	100: (* Done *)
		bDone := (nErrorId = BACnet_ERR_NO_ERROR);
		(* release ADS buffer *)
		stBACnet_AdsBuffer.iLocked := 0;
		(* go idle *)
		_i := 0;

END_CASE

(* set error flag *)
bError 	:= nErrorId > BACnet_ERR_NO_ERROR;
bBusy 	:= _i > 0;
END_FUNCTION_BLOCK
ACTION _NextLogDatum:
_bNextDatum := (_pLrDatumList^.nEntrySize AND 16#80000000) = 16#80000000;
_cbTmpSize := 	(_F_BACnet_AlignedSize(_pLrDatumList^.nEntrySize) AND 16#7FFFFFFF)
			+	SIZEOF(_pLrDatumList^.nEntrySize)
			+	SIZEOF(_pLrDatumList^.reserved);
_pLrDatumList := _pLrDatumList + _cbTmpSize;
END_ACTION
ACTION _NextLogRecord:
_bNextRecord := ((_pLbRecordList^.nEntrySize AND 16#80000000) = 16#80000000);
_cbTmpSize := _F_BACnet_AlignedSize(_pLbRecordList^.nEntrySize AND 16#7FFFFFFF) + SIZEOF(_pLbRecordList^.nEntrySize) + SIZEOF(_pLbRecordList^.nSequence);
_pLbRecordList	:= _pLbRecordList + _cbTmpSize;
_cbTotalBuf := _cbTotalBuf + _cbTmpSize;
END_ACTION

(* POU FB_BACnet_ObjectNameProperty, ST *)
FUNCTION_BLOCK FB_BACnet_ObjectNameProperty
VAR_INPUT
	tObjectID			: T_BACnet_ObjectIdentifier := 16#FFFFFFFF;
	bAutoGet			: BOOL:=TRUE; (* TRUE = get data from property when ADS connection OR object ID changed *)
	bGet				: BOOL; (* FALSE --> TRUE = get data from property *)
END_VAR
VAR_IN_OUT
	stAdsConn			: ST_BACnet_AdsConnection;
END_VAR
VAR_OUTPUT
	bDone				: BOOL;
	bBusy				: BOOL;
	bError				: BOOL;
	nErrorId			: UINT;
	sText				: T_MaxString; (* Object name *)
END_VAR
VAR
	_fbReadProp		: FB_BACnet_ReadProp;
	_i				: INT;
	_rtrigGetSet	: R_TRIG;
	_nAdsReloadOld	: USINT;
	_tObjectIDOld	: T_BACnet_ObjectIdentifier := 16#FFFFFFFF;
	_StringExtDecode: FB_BACnet_StringExtDecode;
END_VAR
(* ADS read *)
_fbReadProp(
	BACnetDevicePort	:= stAdsConn.nAmsPort,
	bExecute			:= ,
	sNetId				:= stAdsConn.sAmsNetId,
	ObjectType			:= F_BACnet_GetObjType(tObjectID),
	PropertyID			:= BACnetPropertyIdentifier_ObjectName,
	DataType			:= BACnetDataType_CharacterStringExt,
	ObjectInstance		:= F_BACnet_GetObjInstance(tObjectID),
	ptrValue			:= ADR(sText),
	nLenValue			:= SIZEOF(sText)-1,
	bDone				=> ,
	bBusy				=> ,
	bError				=> ,
	nErrID				=> ,
	nProcessedLen		=> );

(* trigger start event *)
_rtrigGetSet(CLK:= bGet, Q=> );

(* state machine *)
CASE _i OF

	0: (* Idle *)
		IF		(		(		_rtrigGetSet.Q
							OR	(_nAdsReloadOld <> stAdsConn.nReload)
							OR	(_tObjectIDOld <> tObjectID)
						)
					AND	bAutoGet
				)
			OR	_rtrigGetSet.Q
		THEN
			IF (NOT stAdsConn.bValid) THEN
				(* ADS connection not valid *)
				nErrorId := BACnet_ERR_INVALID_ADS_CONN;
			ELSE
				nErrorId := BACnet_ERR_NO_ERROR;
				_i := 1;
				sText := '';
				(* remind ADS reload counter and parameter *)
				_nAdsReloadOld := stAdsConn.nReload;
				_tObjectIDOld := tObjectID;
			END_IF
			(* reset done flag *)
			bDone := FALSE;
		END_IF
		IF (NOT bGet) AND (NOT bAutoGet) THEN
			nErrorId := BACnet_ERR_NO_ERROR;
			bDone := FALSE;
		END_IF

	(* READ *)
	1: (* read object property data over ADS *)
		IF _fbReadProp.bExecute THEN
			IF _fbReadProp.bError THEN
				_i := 100;
				nErrorId := BACnet_ERR_ADS_Read;
				_fbReadProp.bExecute := FALSE;
			ELSIF (NOT _fbReadProp.bBusy) THEN
				_fbReadProp.bExecute := FALSE;
				(* decode property data *)
				_StringExtDecode(
					pChrStringExt	:= ADR(sText),
					nSize			:= _fbReadProp.nProcessedLen,
					pOutString		:= ADR(sText),
					bValid			=> ,
					bOverflow		=> ,
					nLength			=> ,
					eSrcEncoding	=> );
				(* check overflow flag *)
				IF _StringExtDecode.bOverflow THEN
					nErrorId := BACnet_ERR_ADS_BufferSize;
				END_IF
				(* DONE *)
				_i := 100;
			END_IF
		ELSE
			_fbReadProp.bExecute := TRUE;
		END_IF

	100: (* Done *)
		bDone := (nErrorId = BACnet_ERR_NO_ERROR);
		_i := 0;

END_CASE

(* set error flag *)
bError 	:= nErrorId > BACnet_ERR_NO_ERROR;
bBusy 	:= _i > 0;
END_FUNCTION_BLOCK

(* POU FB_BACnet_Loop, ST *)
FUNCTION_BLOCK FB_BACnet_Loop
VAR_INPUT
	fAccLimit		: REAL := 0.0; (* Setpoint acceleration limit positive and negative [1/s] *)
END_VAR
VAR_IN_OUT
	Device			: FB_BACnet_Device;
END_VAR
VAR_OUTPUT
	bReady			: BOOL;
	fSetPoint		: REAL;
	fControlledValue: REAL;
	fPresentValue	: REAL;
	fPropBand		: REAL; (* controller output in range of -100...100% in relation to Min.-/Max.-output *)
	bOverridden		: BOOL;
	bOutOfService	: BOOL;
	bFault			: BOOL;
	bInAlarm		: BOOL;
	bOpenLoop		: BOOL;
	bCommFailure	: BOOL;
	bOtherFault		: BOOL;
	bError			: BOOL;
	nErrorId		: UINT;
END_VAR
VAR
	_ControlledVariableValue AT%I*: REAL;	(* ~(BACnet_ControlledVariableValue :		: )
												(BACnet_ObjectType				: LOOP	: )	*)
	_Setpoint AT%I*:REAL;					(* ~(BACnet_Setpoint				:		: )	*)
	_ProportionalConstant AT%I*:REAL;		(* ~(BACnet_ProportionalConstant	:		: )	*)
	_IntegralConstant AT%I*:REAL;			(* ~(BACnet_IntegralConstant	 	:		: )	*)
	_DerivativeConstant AT%I*:REAL;			(* ~(BACnet_DerivativeConstant	 	:		: )	*)
	_MaximumOutput AT%I*:REAL;				(* ~(BACnet_MaximumOutput			:		: )	*)
	_MinimumOutput AT%I*:REAL;				(* ~(BACnet_MinimumOutput			:		: )	*)
	_Bias AT%I*:REAL;						(* ~(BACnet_Bias					:		: )	*)
	_PresentValueI AT%I*: REAL; 			(* ~(BACnet_PresentValue 			: 		: )	*)
	_StatusFlags AT%I*: WORD; 				(* ~(BACnet_StatusFlags 			: 		: )	*)
	_Reliability AT%I*: E_BACNETRELIABILITY;(* ~(BACNET_RELIABILITY 			:		: )	*)
	_ControlAction AT%I*:E_BACNETACTION;	(* ~(BACNET_ACTION				 	:		: )	*)
	_PresentValueQ AT%Q*: REAL;				(* ~(BACnet_PresentValue	 		:		: )	*)
	_StatusFlagsBits : ST_BACnet_StatusFlags;

	_sysTime	: GETCPUCOUNTER;
	_Time		: T_LARGE_INTEGER;
	_TimeOld	: T_LARGE_INTEGER;
	_cycleTime	: REAL;
	_PidControl : FB_BACnet_PidControl;
	_fbAccLimit : FB_BACnet_AccLimit;

	_nUpdateCount : UDINT := 0;
END_VAR
(* update server device *)
IF (Device._nUpdateCount = _nUpdateCount) THEN
	Device();
END_IF
(* remind current number of update counter *)
_nUpdateCount := Device._nUpdateCount;

(* determine cycle time *)
_TimeOld := _Time;
_sysTime(cpuCntLoDW=> _Time.dwLowPart, cpuCntHiDW=> _Time.dwHighPart);
_cycleTime := _F_BACnet_SysTimeDiff(In1:=_Time, In2:=_TimeOld);

(* check BitString format of StatusFlags --> if StatusFlags are less than 4, object isn't linked correctly *)
IF (_StatusFlags < 4) THEN
	(* wrong mapping *)
	nErrorId := BACnet_ERR_WRONG_MAPPING;
	bReady := FALSE;

ELSIF Device.bOperational THEN
	(* ready state *)
	bReady := TRUE;
	nErrorId := BACnet_ERR_NO_ERROR;

	(* decode status flags *)
	_StatusFlagsBits := F_BACnet_StatusFlags(_StatusFlags);

	(* copy states to output *)
	bOverridden := _StatusFlagsBits.overridden;
	bOutOfService := _StatusFlagsBits.out_of_service;
	bFault := _StatusFlagsBits.fault;
	bInAlarm := _StatusFlagsBits.in_alarm;
	bOpenLoop := (_Reliability = BACnetReliability_open_loop);
	bCommFailure := (_Reliability = BACnetReliability_communication_failure);
	bOtherFault := (_Reliability = BACnetReliability_unreliable_other);

	(* check reliability *)
	IF _Reliability <> BACnetReliability_no_fault_detected THEN
		_PidControl.bReset			:= TRUE;

	(* is set out of service? *)
	ELSIF _StatusFlagsBits.out_of_service THEN
		_PidControl.bReset			:= TRUE;

	(* decide the control action (direct or reverse) *)
	ELSIF _ControlAction = BACnetAction_direct THEN
		_PidControl.bReset			:= FALSE;
		_PidControl.fPresentValue	:= _ControlledVariableValue;
		_PidControl.fSetpoint		:= _Setpoint;

	ELSIF _ControlAction = BACnetAction_reverse THEN
		_PidControl.bReset			:= FALSE;
		_PidControl.fPresentValue	:= _Setpoint;
		_PidControl.fSetpoint		:= _ControlledVariableValue;

	ELSE
		(* unknown action *)
		_PidControl.bReset			:= TRUE;
	END_IF

	(* call PID control function block *)
	_PidControl(
		fCtrlCycleTime	:= _cycleTime,
		fBias			:= _Bias,
		fKp				:= _ProportionalConstant,
		fKi				:= _IntegralConstant,
		fKd				:= _DerivativeConstant,
		fTp				:= -1.0,
		fMaxOutput		:= _MaximumOutput,
		fMinOutput		:= _MinimumOutput,
		nErrorStatus	=>
	);
	_fbAccLimit.X := _PidControl.fY;

	(* set other outputs *)
	fSetPoint := _Setpoint;
	fPresentValue := _PresentValueI;
	fControlledValue := _ControlledVariableValue;
ELSE
	(* server device not ready, reset local ready also *)
	bReady := FALSE;
	nErrorId := BACnet_ERR_OPERATIONAL;
END_IF

(* limit present value *)
_fbAccLimit(X:= , Amax:= fAccLimit, Tcycle:= _cycleTime, Y=> _PresentValueQ, A=> );

(* calculate proportional band *)
IF (_MaximumOutput > 0.0) AND (_MinimumOutput >= 0.0) THEN
	fPropBand := ((_PresentValueQ - _MinimumOutput) / (_MaximumOutput - _MinimumOutput)) * 100.0;
ELSIF (_MaximumOutput <= 0.0) AND (_MinimumOutput < 0.0) THEN
	fPropBand := ((_PresentValueQ - _MaximumOutput) / (_MaximumOutput - _MinimumOutput)) * 100.0;
ELSIF (_PresentValueQ > 0.0) AND (_MaximumOutput > 0.0) THEN
	fPropBand := (_PresentValueQ / _MaximumOutput) * 100.0;
ELSIF (_PresentValueQ < 0.0) AND (_MinimumOutput < 0.0) THEN
	fPropBand := (_PresentValueQ / _MinimumOutput) * -100.0;
ELSE
	fPropBand := 0.0;
END_IF

(* set error flag *)
bError := (nErrorId <> BACnet_ERR_NO_ERROR);
END_FUNCTION_BLOCK

(* POU FB_BACnet_PidControl, ST *)
FUNCTION_BLOCK FB_BACnet_PidControl
VAR_INPUT
	(* controller input  *)
	fSetpoint				: REAL;	(* setpoint value *)
	fPresentValue			: REAL;	(* actual value *)
	(* reset flag *)
	bReset					: BOOL;
	(* controller values *)
	fCtrlCycleTime			: REAL; (* controller cycle time in seconds [s] *)

	fBias					: REAL; (* bias also active when reset is set to 1 *)
	fKp						: REAL;	(* proportional gain Kp	(P) *)
	fKi						: REAL; (* integral gain Ki (I) *)
	fKd						: REAL;	(* derivative gain Kd (D) *)
	fTp						: REAL := -1.0;	(* damping time Tp (PT1) [s] (fTp < 0 --> Tp = Kd / 10) *)

	(* maximum ratings *)
	fMaxOutput				: REAL;
	fMinOutput				: REAL;
END_VAR
VAR_OUTPUT
	fY						: REAL; (* controller output command *)
	nErrorStatus			: UINT; (* controller error output (0: no error; >0:error) *)
END_VAR
VAR
	(* Internal Variable *)
	_fE		: REAL;
	_fEOld	: REAL;
	_fYp	: REAL;
	_fYi	: REAL;
	_fYd	: REAL;
	_fbYd	: FB_BACnet_PT1;
END_VAR
(* preset error number *)
nErrorStatus	:= BACnet_ERR_NO_ERROR;

(* check cycle time parameter: (CycleTime > 0) *)
IF (fCtrlCycleTime <= 0.0) THEN
	nErrorStatus := BACnet_ERR_INVALID_CYCLETIME;
	bReset := TRUE;
END_IF;

(* check controller parameters: (Kp, Ki, Kd >= 0) *)
IF ((fKp < 0.0) OR (fKi < 0.0) OR (fKd < 0.0)) THEN
	nErrorStatus := BACnet_ERR_INVALID_PARAMETER;
	bReset := TRUE;
END_IF;

(* controller reset *)
IF bReset THEN
	(* reset internal and external variables *)
	_fEOld	:= 0.0;
	fY		:= MAX(MIN(fBias, fMaxOutput), fMinOutput);
	_fYi	:= 0.0;
	_fbYd(X:= 0.0, T:= 0.0, Y=> );
	RETURN;
END_IF

(* 3. save old variable *)
_fEOld := _fE;

(* 4. set error/deviation input *)
_fE := fSetpoint - fPresentValue;

(* 5. YP-part *)
_fYp := fKp * _fE;

(* 6. YI-part *)
IF (fKi = 0.0) THEN
	_fYi	:= 0.0;
ELSE
	_fYi := _fYi + (fKi * fCtrlCycleTime * _fE);
END_IF
IF (_fYi > fMaxOutput) THEN
	(* limit wind up positive *)
	_fYi := fMaxOutput;
ELSIF (_fYi < fMinOutput) THEN
	(* limit wind up negative *)
	_fYi := fMinOutput;
END_IF

(* 7. YD-part *)
IF (fTp < 0.0) THEN
	fTp := fKd / 10.0;
END_IF
_fYd := fKd * (_fE - _fEOld) / fCtrlCycleTime;
_fbYd(X:= _fYd, T:= fTp, Tcycle:= fCtrlCycleTime, Y=> );

(* 8. Ysum = YP + YI + YD + Bias and output *)
fY := _fYp + _fYi + _fbYd.Y + fBias;
fY := MAX(MIN(fY, fMaxOutput), fMinOutput);
END_FUNCTION_BLOCK

(* POU FB_BACnet_Loop_DRV, ST *)
FUNCTION_BLOCK FB_BACnet_Loop_DRV
VAR_IN_OUT
	Device	: FB_BACnet_Device;
END_VAR
VAR_OUTPUT
	bReady				: BOOL;
	fSetPoint			: REAL;
	fControlledValue	: REAL;
	fPresentValue		: REAL;
	bOverridden			: BOOL;
	bOutOfService		: BOOL;
	bFault				: BOOL;
	bInAlarm			: BOOL;
	bError				: BOOL;
	nErrorId			: UINT;
END_VAR
VAR
	_ControlledVariableValue AT%I*: REAL;	(* ~(BACnet_ControlledVariableValue :		: )
												(BACnet_ObjectType				: LOOP	: )
												(BACnet_EnableInternalLoopCtrl	: TRUE	: NOLINK,ENABLE) *)
	_Setpoint AT%I*:REAL;					(* ~(BACnet_Setpoint				:		: )	*)
	_PresentValue AT%I*: REAL; 				(* ~(BACnet_PresentValue 			: 		: )	*)
	_ObjectId AT%I*: DWORD;					(* ~(BACnet_ObjectIdentifier		:		: LINK) *)
	_StatusFlags AT%I*: WORD; 				(* ~(BACnet_StatusFlags 			: 		: )	*)
	_StatusFlagsBits : ST_BACnet_StatusFlags;
	_nUpdateCount : UDINT := 0;
END_VAR
(* update server device *)
IF (Device._nUpdateCount = _nUpdateCount) THEN
	Device();
END_IF
(* remind current number of update counter *)
_nUpdateCount := Device._nUpdateCount;

(* check BitString format of StatusFlags --> if StatusFlags are less than 4, object isn't linked correctly *)
IF (_StatusFlags < 4) THEN
	(* wrong mapping *)
	nErrorId := BACnet_ERR_WRONG_MAPPING;
	bReady := FALSE;

ELSIF Device.bOperational THEN
	(* ready state *)
	bReady := TRUE;
	nErrorId := BACnet_ERR_NO_ERROR;

	(* decode status flags *)
	_StatusFlagsBits := F_BACnet_StatusFlags(_StatusFlags);

	(* copy states to output *)
	bOverridden := _StatusFlagsBits.overridden;
	bOutOfService := _StatusFlagsBits.out_of_service;
	bFault := _StatusFlagsBits.fault;
	bInAlarm := _StatusFlagsBits.in_alarm;

	(* set other outputs *)
	fSetPoint := _Setpoint;
	fPresentValue := _PresentValue;
	fControlledValue := _ControlledVariableValue;
ELSE
	(* server device not ready, reset local ready also *)
	bReady := FALSE;
	nErrorId := BACnet_ERR_OPERATIONAL;
END_IF
(* set error flag *)
bError := (nErrorId <> BACnet_ERR_NO_ERROR);
END_FUNCTION_BLOCK

(* POU FB_BACnet_Loop_DRV_EX, ST *)
FUNCTION_BLOCK FB_BACnet_Loop_DRV_EX
VAR_IN_OUT
	Device	: FB_BACnet_Device;
END_VAR
VAR_OUTPUT
	bReady				: BOOL;
	fSetPoint			: REAL;
	fControlledValue	: REAL;
	fPresentValue		: REAL;
	fPropBand			: REAL; (* controller output in range of -100...100% in relation to Min.-/Max.-output *)
	bOverridden			: BOOL;
	bOutOfService		: BOOL;
	bFault				: BOOL;
	bInAlarm			: BOOL;
	bOpenLoop			: BOOL;
	bCommFailure		: BOOL;
	bOtherFault			: BOOL;
	eEventState			: E_BACNETEVENTSTATE;
	bAckedTrans_ToOffNormal : BOOL;
	bAckedTrans_ToFault		: BOOL;
	bAckedTrans_ToNormal	: BOOL;
	tObjectID			: T_BACnet_ObjectIdentifier := 16#FFFFFFFF;
	bError				: BOOL;
	nErrorId			: UINT;
END_VAR
VAR
	_ControlledVariableValue AT%I*: REAL;	(* ~(BACnet_ControlledVariableValue :		: )
												(BACnet_ObjectType				: LOOP	: )
												(BACnet_EnableInternalLoopCtrl	: TRUE	: NOLINK,ENABLE) *)
	_Setpoint AT%I*:REAL;					(* ~(BACnet_Setpoint				:		: )	*)
	_MaximumOutput AT%I*:REAL;				(* ~(BACnet_MaximumOutput			:		: )	*)
	_MinimumOutput AT%I*:REAL;				(* ~(BACnet_MinimumOutput			:		: )	*)
	_PresentValue AT%I*: REAL; 				(* ~(BACnet_PresentValue 			: 		: )	*)
	_ObjectId AT%I*: DWORD;					(* ~(BACnet_ObjectIdentifier		:		: LINK) *)
	_StatusFlags AT%I*: WORD; 				(* ~(BACnet_StatusFlags 			: 		: )	*)
	_AckedTransitions AT%I*:WORD;			(* ~(BACnet_AckedTransitions		:		: ) *)
	_EventState AT%I*: WORD; 				(* ~(BACnet_EventState 				:		: )	*)
	_Reliability AT%I*: E_BACNETRELIABILITY;(* ~(BACNET_RELIABILITY 			:		: )	*)
	_StatusFlagsBits : ST_BACnet_StatusFlags;
	_AckedTransBits : ST_BACnet_EventTransitionBits;
	_nUpdateCount : UDINT := 0;
END_VAR
(* update server device *)
IF (Device._nUpdateCount = _nUpdateCount) THEN
	Device();
END_IF
(* remind current number of update counter *)
_nUpdateCount := Device._nUpdateCount;

(* check BitString format of StatusFlags --> if StatusFlags are less than 4, object isn't linked correctly *)
IF (F_BACnet_GetObjType(_ObjectId) <> BACnetObjectType_Loop) THEN
	(* wrong mapping / invalid object ID *)
	IF _ObjectId = 0 THEN
		nErrorId := BACnet_ERR_WRONG_MAPPING;
	ELSE
		nErrorId := BACnet_ERR_INVALID_OBJECTID;
	END_IF
	bReady := FALSE;
	tObjectID := 16#FFFFFFFF;

ELSIF (_StatusFlags < 4) OR _AckedTransitions < 5 THEN
	(* wrong mapping *)
	nErrorId := BACnet_ERR_WRONG_MAPPING;
	bReady := FALSE;

ELSIF Device.bOperational THEN
	(* ready state *)
	bReady := TRUE;
	nErrorId := BACnet_ERR_NO_ERROR;

	(* decode status flags *)
	_StatusFlagsBits := F_BACnet_StatusFlags(_StatusFlags);
	_AckedTransBits	:= F_BACnet_EventTransitionFlags(_AckedTransitions);

	(* copy states to output *)
	bOverridden := _StatusFlagsBits.overridden;
	bOutOfService := _StatusFlagsBits.out_of_service;
	bFault := _StatusFlagsBits.fault;
	bInAlarm := _StatusFlagsBits.in_alarm;
	bOpenLoop := (_Reliability = BACnetReliability_open_loop);
	bCommFailure := (_Reliability = BACnetReliability_communication_failure);
	bOtherFault := (_Reliability = BACnetReliability_unreliable_other);
	bAckedTrans_ToOffNormal := _AckedTransBits.to_offnormal;
	bAckedTrans_ToFault := _AckedTransBits.to_fault;
	bAckedTrans_ToNormal := _AckedTransBits.to_normal;
	tObjectID := _ObjectId;
	eEventState := _EventState;

	(* calculate proportional band *)
	IF (_MaximumOutput > 0.0) AND (_MinimumOutput >= 0.0) THEN
		fPropBand := ((_PresentValue - _MinimumOutput) / (_MaximumOutput - _MinimumOutput)) * 100.0;
	ELSIF (_MaximumOutput <= 0.0) AND (_MinimumOutput < 0.0) THEN
		fPropBand := ((_PresentValue - _MaximumOutput) / (_MaximumOutput - _MinimumOutput)) * 100.0;
	ELSIF (_PresentValue > 0.0) AND (_MaximumOutput > 0.0) THEN
		fPropBand := (_PresentValue / _MaximumOutput) * 100.0;
	ELSIF (_PresentValue < 0.0) AND (_MinimumOutput < 0.0) THEN
		fPropBand := (_PresentValue / _MinimumOutput) * -100.0;
	ELSE
		fPropBand := 0.0;
	END_IF

	(* set other outputs *)
	fSetPoint := _Setpoint;
	fPresentValue := _PresentValue;
	fControlledValue := _ControlledVariableValue;
ELSE
	(* server device not ready, reset local ready also *)
	bReady := FALSE;
	nErrorId := BACnet_ERR_OPERATIONAL;
END_IF
(* set error flag *)
bError := (nErrorId <> BACnet_ERR_NO_ERROR);
END_FUNCTION_BLOCK

(* POU FB_BACnet_Loop_EX, ST *)
FUNCTION_BLOCK FB_BACnet_Loop_EX
VAR_INPUT
	bAutoTuning			: BOOL; (* Start autotuning of PID controller *)
	tTuningTimeout		: TIME := T#15m; (* Maximum runtime of tuning procedure [ms] *)
	eTuningMode			: E_BACNETPIDTUNINGMODE := BACnetPIDTuningMode_PI; (* optimize default PI controller *)
	fAccLimit			: REAL := 0.0; (* Setpoint acceleration limit positive and negative [1/s] *)
END_VAR
VAR_IN_OUT
	Device				: FB_BACnet_Device;
END_VAR
VAR_OUTPUT
	bReady				: BOOL;
	bTuningActive		: BOOL;
	bTuningWaitPV		: BOOL;
	bTuningWaitCV		: BOOL;
	bTuningDone			: BOOL;
	bTuningAborted		: BOOL;
	fSetPoint			: REAL;
	fControlledValue	: REAL;
	fPresentValue		: REAL;
	fPropBand			: REAL; (* controller output in range of -100...100% in relation to Min.-/Max.-output *)
	bOverridden			: BOOL;
	bOutOfService		: BOOL;
	bFault				: BOOL;
	bInAlarm			: BOOL;
	bOpenLoop			: BOOL;
	bCommFailure		: BOOL;
	bOtherFault			: BOOL;
	eEventState			: E_BACNETEVENTSTATE;
	bAckedTrans_ToOffNormal : BOOL;
	bAckedTrans_ToFault		: BOOL;
	bAckedTrans_ToNormal	: BOOL;
	tObjectID			: T_BACnet_ObjectIdentifier := 16#FFFFFFFF;
	bError				: BOOL;
	nErrorId			: UINT;
END_VAR
VAR
	_ControlledVariableValue AT%I*: REAL;	(* ~(BACnet_ControlledVariableValue :		: )
												(BACnet_ObjectType				: LOOP	: )	*)
	_Setpoint AT%I*:REAL;					(* ~(BACnet_Setpoint				:		: )	*)
	_ProportionalConstant AT%I*:REAL;		(* ~(BACnet_ProportionalConstant	:		: )	*)
	_IntegralConstant AT%I*:REAL;			(* ~(BACnet_IntegralConstant	 	:		: )	*)
	_DerivativeConstant AT%I*:REAL;			(* ~(BACnet_DerivativeConstant	 	:		: )	*)
	_MaximumOutput AT%I*:REAL;				(* ~(BACnet_MaximumOutput			:		: )	*)
	_MinimumOutput AT%I*:REAL;				(* ~(BACnet_MinimumOutput			:		: )	*)
	_Bias AT%I*:REAL;						(* ~(BACnet_Bias					:		: )	*)
	_PresentValueI AT%I*: REAL; 			(* ~(BACnet_PresentValue 			: 		: )	*)
	_Deadband AT%I*: REAL; 					(* ~(BACnet_Deadband	 			: 		: )	*)
	_ObjectId AT%I*: DWORD;					(* ~(BACnet_ObjectIdentifier		:		: LINK) *)
	_StatusFlags AT%I*: WORD; 				(* ~(BACnet_StatusFlags 			: 		: )	*)
	_AckedTransitions AT%I*:WORD;			(* ~(BACnet_AckedTransitions		:		: ) *)
	_EventState AT%I*: WORD; 				(* ~(BACnet_EventState 				:		: )	*)
	_Reliability AT%I*: E_BACNETRELIABILITY;(* ~(BACNET_RELIABILITY 			:		: )	*)
	_ControlAction AT%I*:E_BACNETACTION;	(* ~(BACNET_ACTION				 	:		: )	*)
	_PresentValueQ AT%Q*: REAL;				(* ~(BACnet_PresentValue	 		:		: )	*)
	_AckedTransBits : ST_BACnet_EventTransitionBits;
	_StatusFlagsBits : ST_BACnet_StatusFlags;

	_sysTime	: GETCPUCOUNTER;
	_Time		: T_LARGE_INTEGER;
	_TimeOld	: T_LARGE_INTEGER;
	_cycleTime	: REAL;
	_PidControl : FB_BACnet_PidControl;
	_AutoTuning : _FB_BACnet_PidTune;
	_iTuning	: INT;
	_WriteProp	: FB_BACnet_WriteProp;
	_fbAccLimit : FB_BACnet_AccLimit;
	_nUpdateCount : UDINT := 0;
END_VAR
(* update server device *)
IF (Device._nUpdateCount = _nUpdateCount) THEN
	Device();
END_IF
(* remind current number of update counter *)
_nUpdateCount := Device._nUpdateCount;

(* determine cycle time *)
_TimeOld := _Time;
_sysTime(cpuCntLoDW=> _Time.dwLowPart, cpuCntHiDW=> _Time.dwHighPart);
_cycleTime := _F_BACnet_SysTimeDiff(In1:=_Time, In2:=_TimeOld);

(* check BitString format of StatusFlags --> if StatusFlags are less than 4, object isn't linked correctly *)
IF (F_BACnet_GetObjType(_ObjectId) <> BACnetObjectType_Loop) THEN
	(* wrong mapping / invalid object ID *)
	IF _ObjectId = 0 THEN
		nErrorId := BACnet_ERR_WRONG_MAPPING;
	ELSE
		nErrorId := BACnet_ERR_INVALID_OBJECTID;
	END_IF
	bReady := FALSE;
	tObjectID := 16#FFFFFFFF;

ELSIF (_StatusFlags < 4) OR _AckedTransitions < 5 THEN
	(* wrong mapping *)
	nErrorId := BACnet_ERR_WRONG_MAPPING;
	bReady := FALSE;

ELSIF Device.bOperational THEN
	(* ready state *)
	bReady := TRUE;
	nErrorId := BACnet_ERR_NO_ERROR;

	(* decode status flags *)
	_StatusFlagsBits := F_BACnet_StatusFlags(_StatusFlags);
	_AckedTransBits	:= F_BACnet_EventTransitionFlags(_AckedTransitions);

	(* copy states to output *)
	bOverridden := _StatusFlagsBits.overridden;
	bOutOfService := _StatusFlagsBits.out_of_service;
	bFault := _StatusFlagsBits.fault;
	bInAlarm := _StatusFlagsBits.in_alarm;
	bOpenLoop := (_Reliability = BACnetReliability_open_loop);
	bCommFailure := (_Reliability = BACnetReliability_communication_failure);
	bOtherFault := (_Reliability = BACnetReliability_unreliable_other);
	bAckedTrans_ToOffNormal := _AckedTransBits.to_offnormal;
	bAckedTrans_ToFault := _AckedTransBits.to_fault;
	bAckedTrans_ToNormal := _AckedTransBits.to_normal;
	tObjectID := _ObjectId;
	eEventState := _EventState;

	(* check if auto tuning is active *)
	IF bTuningActive THEN
		_PidControl.bReset			:= TRUE;

	(* check reliability *)
	ELSIF _Reliability <> BACnetReliability_no_fault_detected THEN
		_PidControl.bReset			:= TRUE;

	(* is set out of service? *)
	ELSIF _StatusFlagsBits.out_of_service THEN
		_PidControl.bReset			:= TRUE;

	(* decide the control action (direct or reverse) *)
	ELSIF _ControlAction = BACnetAction_direct THEN
		_PidControl.bReset			:= FALSE;
		_PidControl.fPresentValue	:= _ControlledVariableValue;
		_PidControl.fSetpoint		:= _Setpoint;

	ELSIF _ControlAction = BACnetAction_reverse THEN
		_PidControl.bReset			:= FALSE;
		_PidControl.fPresentValue	:= _Setpoint;
		_PidControl.fSetpoint		:= _ControlledVariableValue;

	ELSE
		(* unknown action *)
		_PidControl.bReset			:= TRUE;
	END_IF

	(* call PID control function block *)
	_PidControl(
		fCtrlCycleTime	:= _cycleTime,
		fBias			:= _Bias,
		fKp				:= _ProportionalConstant,
		fKi				:= _IntegralConstant,
		fKd				:= _DerivativeConstant,
		fTp				:= -1.0,
		fMaxOutput		:= _MaximumOutput,
		fMinOutput		:= _MinimumOutput,
		nErrorStatus	=>
	);
	IF (_iTuning < 10) THEN
		_fbAccLimit.X := _PidControl.fY;
	END_IF

	(* set other outputs *)
	fSetPoint := _Setpoint;
	fPresentValue := _PresentValueI;
	fControlledValue := _ControlledVariableValue;
ELSE
	(* server device not ready, reset local ready also *)
	bReady := FALSE;
	nErrorId := BACnet_ERR_OPERATIONAL;
END_IF

(* write controller settings *)
_WriteProp.BACnetDevicePort:= Device.stAdsConn.nAmsPort;
_WriteProp.sNetId		:= Device.stAdsConn.sAmsNetId;
_WriteProp.ObjectType	:= BACnetObjectType_Loop;
_WriteProp.ObjectInstance:= F_BACnet_GetObjInstance(_ObjectId);

(* Autotuning function *)
CASE _iTuning OF
	0: (* Idle *)
		IF		bReady						(* object ready *)
			AND	(NOT _PidControl.bReset)	(* PID controller ready *)
			AND (tTuningTimeout > t#0ms)	(* timeout valid *)
			AND bAutoTuning					(* start flag *)
		THEN
			_iTuning := 5;
		END_IF
		_AutoTuning.bStart := FALSE;

	5:
		(* present_value low *)
		IF (_PresentValueI <= ((_MaximumOutput + _MinimumOutput) / 2.0) + _Bias) THEN
			_iTuning := 10;
		ELSIF (NOT bAutoTuning) THEN
			_iTuning := 0;
		END_IF

	10: (* setup *)
		_AutoTuning.fSetY	:= _MaximumOutput;
		_AutoTuning.tTimeout:= tTuningTimeout;
		_AutoTuning.fMinY	:= _MinimumOutput;
		_AutoTuning.fMaxY	:= _MaximumOutput;
		_AutoTuning.fDeadband:= _Deadband;
		_AutoTuning.eMode	:= eTuningMode;
		_iTuning := 20;

	20: (* wait busy *)
		_AutoTuning.bStart := TRUE;
		IF _AutoTuning.bAborted THEN
			_iTuning := 200;
		ELSIF _AutoTuning.bBusy THEN
			_iTuning := 30;
		END_IF

	30: (* wait done *)
		IF _AutoTuning.bAborted THEN
			_iTuning := 200;
		ELSIF _AutoTuning.bDone THEN
			_iTuning := 40;
		END_IF

	40: (* write properties *)
		IF Device.stAdsConn.bValid THEN
			_iTuning := 41;
			_WriteProp(bExecute := FALSE);
		ELSE
			_iTuning := 200;
		END_IF

	41: (* write Kp *)
		_WriteProp.DataType	:= BACnetDataType_Real;
		_WriteProp.ptrValue	:= ADR(_AutoTuning.fPID_Kp);
		_WriteProp.nLenValue:= SIZEOF(_AutoTuning.fPID_Kp);
		_WriteProp(
			bExecute := TRUE,
			PropertyID := BACnetPropertyIdentifier_ProportionalConstant);
		IF (NOT _WriteProp.bBusy) THEN
			IF (_WriteProp.bError) THEN
				_iTuning := 200;
			ELSE
				_iTuning := 42;
			END_IF
			_WriteProp(bExecute := FALSE);
		END_IF

	42: (* write Ki *)
		_WriteProp.DataType	:= BACnetDataType_Real;
		_WriteProp.ptrValue	:= ADR(_AutoTuning.fPID_Ki);
		_WriteProp.nLenValue:= SIZEOF(_AutoTuning.fPID_Ki);
		_WriteProp(
			bExecute := TRUE,
			PropertyID := BACnetPropertyIdentifier_IntegralConstant);
		IF (NOT _WriteProp.bBusy) THEN
			IF (_WriteProp.bError) THEN
				_iTuning := 200;
			ELSE
				_iTuning := 43;
			END_IF
			_WriteProp(bExecute := FALSE);
		END_IF

	43: (* write Kd *)
		_WriteProp.DataType	:= BACnetDataType_Real;
		_WriteProp.ptrValue	:= ADR(_AutoTuning.fPID_Kd);
		_WriteProp.nLenValue:= SIZEOF(_AutoTuning.fPID_Kd);
		_WriteProp(
			bExecute := TRUE,
			PropertyID := BACnetPropertyIdentifier_DerivativeConstant);
		IF (NOT _WriteProp.bBusy) THEN
			IF (_WriteProp.bError) THEN
				_iTuning := 200;
			ELSE
				_iTuning := 44;
			END_IF
			_WriteProp(bExecute := FALSE);
		END_IF

	44: (* write Action *)
		_WriteProp.DataType	:= BACnetDataType_Enumerated;
		_WriteProp.ptrValue	:= ADR(_AutoTuning.eAction);
		_WriteProp.nLenValue:= SIZEOF(_AutoTuning.eAction);
		_WriteProp(
			bExecute := TRUE,
			PropertyID := BACnetPropertyIdentifier_Action);
		IF (NOT _WriteProp.bBusy) THEN
			IF (_WriteProp.bError) THEN
				_iTuning := 200;
			ELSE
				_iTuning := 100;
			END_IF
			_WriteProp(bExecute := FALSE);
		END_IF


	100: (* done *)
		IF NOT bAutoTuning THEN
			_iTuning := 0;
		END_IF

	200: (* aborted *)
		IF NOT bAutoTuning THEN
			_iTuning := 0;
		END_IF

END_CASE

(* call auto tuning function block *)
_AutoTuning(
	bStart	:= ,
	bStop	:=	_StatusFlagsBits.out_of_service
			OR	(_Reliability <> BACnetReliability_no_fault_detected),
	fSetY	:= ,
	fDeadband	:= ,
	fX		:= _ControlledVariableValue,
	tTimeout:= ,
	fMinY	:= ,
	fMaxY	:= ,
	fCycleTime := _cycleTime,
	fY		:= _fbAccLimit.X,
	fPID_Kp	=> ,
	fPID_Ki	=> ,
	fPID_Kd	=> ,
	eAction => ,
	bSetY	=> ,
	bWaitY	=> ,
	bWaitX	=> ,
	bReady	=> ,
	bBusy	=> ,
	bDone	=> ,
	bAborted=> bTuningAborted,
	bTimeout=> );

(* set auto tuning state *)
bTuningWaitPV	:= (_iTuning = 5);
bTuningWaitCV	:= (_iTuning > 5 AND _iTuning <= 30);
bTuningAborted	:= (_iTuning = 200);
bTuningActive	:= (_iTuning > 0) AND (NOT bTuningAborted);
bTuningDone		:= (_iTuning = 100);
(* set error info *)
IF (bTuningActive OR bTuningAborted) THEN
	IF (NOT Device.stAdsConn.bValid) THEN
		nErrorId	:= BACnet_ERR_INVALID_ADS_CONN;
	ELSIF _WriteProp.bError THEN
		nErrorId	:= BACnet_ERR_ADS_Write;
	END_IF
END_IF

(* limit present value *)
_fbAccLimit(
	X	:= ,
	Amax:= fAccLimit,
	Tcycle:= _cycleTime,
	Y	=> _PresentValueQ,
	A	=> );

(* calculate proportional band *)
IF (_MaximumOutput > 0.0) AND (_MinimumOutput >= 0.0) THEN
	fPropBand := ((_PresentValueQ - _MinimumOutput) / (_MaximumOutput - _MinimumOutput)) * 100.0;
ELSIF (_MaximumOutput <= 0.0) AND (_MinimumOutput < 0.0) THEN
	fPropBand := ((_PresentValueQ - _MaximumOutput) / (_MaximumOutput - _MinimumOutput)) * 100.0;
ELSIF (_PresentValueQ > 0.0) AND (_MaximumOutput > 0.0) THEN
	fPropBand := (_PresentValueQ / _MaximumOutput) * 100.0;
ELSIF (_PresentValueQ < 0.0) AND (_MinimumOutput < 0.0) THEN
	fPropBand := (_PresentValueQ / _MinimumOutput) * -100.0;
ELSE
	fPropBand := 0.0;
END_IF

(* set error flag *)
bError := (nErrorId <> BACnet_ERR_NO_ERROR);
END_FUNCTION_BLOCK

(* POU FB_BACnet_MultiStateInput, ST *)
FUNCTION_BLOCK FB_BACnet_MultiStateInput
VAR_IN_OUT
	Device	: FB_BACnet_Device;
END_VAR
VAR_OUTPUT
	bReady			: BOOL;
	nPresentValue	: UDINT;
	bOverridden		: BOOL;
	bOutOfService	: BOOL;
	bFault			: BOOL;
	bInAlarm		: BOOL;
	bError			: BOOL;
	nErrorId		: UINT;
END_VAR
VAR
	_PresentValue AT%I*: UDINT; 	(* ~(BACnet_PresentValue 	:		: )
								   		(BACnet_ObjectType 		: MI	: )	*)
	_StatusFlags AT%I*: WORD; 		(* ~(BACnet_StatusFlags 	:		: )	*)
	_StatusFlagsBits : ST_BACnet_StatusFlags;

	_nUpdateCount : UDINT := 0;
END_VAR
(* update server device *)
IF (Device._nUpdateCount = _nUpdateCount) THEN
	Device();
END_IF
(* remind current number of update counter *)
_nUpdateCount := Device._nUpdateCount;

(* check BitString format of StatusFlags --> if StatusFlags are less than 4, object isn't linked correctly *)
IF (_StatusFlags < 4) THEN
	(* wrong mapping *)
	nErrorId := BACnet_ERR_WRONG_MAPPING;
	bReady := FALSE;

ELSIF Device.bOperational THEN
	(* ready state *)
	bReady := TRUE;
	nErrorId := BACnet_ERR_NO_ERROR;

	(* present value *)
	nPresentValue := _PresentValue;

	(* build bit states *)
	_StatusFlagsBits := F_BACnet_StatusFlags(_StatusFlags);

	(* copy states to output *)
	bOverridden := _StatusFlagsBits.overridden;
	bOutOfService := _StatusFlagsBits.out_of_service;
	bFault := _StatusFlagsBits.fault;
	bInAlarm := _StatusFlagsBits.in_alarm;

ELSE
	(* server device not ready, reset local ready also *)
	bReady := FALSE;
	nErrorId := BACnet_ERR_OPERATIONAL;
END_IF
(* set error flag *)
bError := (nErrorId <> BACnet_ERR_NO_ERROR);
END_FUNCTION_BLOCK

(* POU FB_BACnet_MultiStateInput_EX, ST *)
FUNCTION_BLOCK FB_BACnet_MultiStateInput_EX
VAR_IN_OUT
	Device				: FB_BACnet_Device;
END_VAR
VAR_OUTPUT
	bReady				: BOOL;
	nPresentValue		: UDINT;
	bOverridden			: BOOL;
	bOutOfService		: BOOL;
	bFault				: BOOL;
	bInAlarm			: BOOL;
	bOverRange			: BOOL;
	bUnderRange			: BOOL;
	bNoSensor			: BOOL;
	bOpenLoop			: BOOL;
	bShortedLoop		: BOOL;
	bMultiStateFault	: BOOL;
	bOtherFault			: BOOL;
	eEventState			: E_BACNETEVENTSTATE;
	bAckedTrans_ToOffNormal : BOOL;
	bAckedTrans_ToFault		: BOOL;
	bAckedTrans_ToNormal	: BOOL;
	nNbrOfStates		: UDINT;
	tObjectID			: T_BACnet_ObjectIdentifier := 16#FFFFFFFF;
	bError				: BOOL;
	nErrorId			: UINT;
END_VAR
VAR
	_PresentValue AT%I*: UDINT; 		(* ~(BACnet_PresentValue 	:		: )
								   			(BACnet_ObjectType 		: MI	: )	*)
	_NumberOfStates AT%I*: UDINT;		(* ~(BACnet_NumberOfStates	:		: )	*)
	_ObjectId AT%I*: DWORD;				(* ~(BACnet_ObjectIdentifier:		: LINK) *)
	_StatusFlags AT%I*: WORD; 			(* ~(BACnet_StatusFlags 	:		: )	*)
	_EventState AT%I*: WORD; 			(* ~(BACnet_EventState 		:		: )	*)
	_Reliability AT%I*: WORD; 			(* ~(BACnet_Reliability 	:		: )	*)
	_AckedTransitions AT%I*:WORD;		(* ~(BACnet_AckedTransitions:		: ) *)
	_AckedTransBits : ST_BACnet_EventTransitionBits;
	_nUpdateCount : UDINT := 0;
	_StatusFlagsBits : ST_BACnet_StatusFlags;
END_VAR
(* update server device *)
IF (Device._nUpdateCount = _nUpdateCount) THEN
	Device();
END_IF
(* remind current number of update counter *)
_nUpdateCount := Device._nUpdateCount;

(* check object type *)
IF (F_BACnet_GetObjType(_ObjectId) <> BACnetObjectType_MultiStateInput) THEN
	(* wrong mapping / invalid object ID *)
	IF _ObjectId = 0 THEN
		nErrorId := BACnet_ERR_WRONG_MAPPING;
	ELSE
		nErrorId := BACnet_ERR_INVALID_OBJECTID;
	END_IF
	bReady := FALSE;

ELSIF (_StatusFlags < 4) OR _AckedTransitions < 5 THEN
	(* wrong mapping *)
	nErrorId := BACnet_ERR_WRONG_MAPPING;
	bReady := FALSE;

ELSIF Device.bOperational THEN
	(* ready state *)
	bReady := TRUE;
	nErrorId := BACnet_ERR_NO_ERROR;

	(* present value *)
	nPresentValue := _PresentValue;

	(* build bit states *)
	_StatusFlagsBits := F_BACnet_StatusFlags(_StatusFlags);
	_AckedTransBits		:= F_BACnet_EventTransitionFlags(_AckedTransitions);

	(* copy states to output *)
	bOverridden := _StatusFlagsBits.overridden;
	bOutOfService := _StatusFlagsBits.out_of_service;
	bFault := _StatusFlagsBits.fault;
	bInAlarm := _StatusFlagsBits.in_alarm;
	bOverRange := (_Reliability = BACnetReliability_over_range);
	bUnderRange := (_Reliability = BACnetReliability_under_range);
	bNoSensor := (_Reliability = BACnetReliability_no_sensor);
	bOpenLoop := (_Reliability = BACnetReliability_open_loop);
	bShortedLoop := (_Reliability = BACnetReliability_shorted_loop);
	bMultiStateFault := (_Reliability = BACnetReliability_multi_state_fault);
	bOtherFault := (_Reliability = BACnetReliability_unreliable_other);
	bAckedTrans_ToOffNormal := _AckedTransBits.to_offnormal;
	bAckedTrans_ToFault := _AckedTransBits.to_fault;
	bAckedTrans_ToNormal := _AckedTransBits.to_normal;
	tObjectID := _ObjectId;

	(* convert enumeration *)
	eEventState := _EventState;

	(* number of states *)
	nNbrOfStates := _NumberOfStates;

ELSE
	(* server device not ready, reset local ready also *)
	bReady := FALSE;
	nErrorId := BACnet_ERR_OPERATIONAL;
END_IF
(* set error flag *)
bError := (nErrorId <> BACnet_ERR_NO_ERROR);
END_FUNCTION_BLOCK

(* POU FB_BACnet_MultiStateInput_RAW, ST *)
FUNCTION_BLOCK FB_BACnet_MultiStateInput_RAW
VAR_INPUT
	nRawIn				AT%Q*: DWORD; (* ~(BACnet_PresentValue : : ) *)
	bNoSensor		: BOOL;
	bOverRange		: BOOL;
	bUnderRange		: BOOL;
	bOpenLoop		: BOOL;
	bShortedLoop	: BOOL;
	bCommFailure	: BOOL;
	bOtherFault		: BOOL;
END_VAR
VAR_IN_OUT
	Device				: FB_BACnet_Device;
END_VAR
VAR_OUTPUT
	bReady				: BOOL;
	nPresentValue		: UDINT;
	bOverridden			: BOOL;
	bOutOfService		: BOOL;
	bFault				: BOOL;
	bInAlarm			: BOOL;
	bAckedTrans_ToOffNormal : BOOL;
	bAckedTrans_ToFault		: BOOL;
	bAckedTrans_ToNormal	: BOOL;
	nNbrOfStates		: UDINT;
	bError				: BOOL;
	nErrorId			: UINT;
END_VAR
VAR
	_Reliability AT%Q*: WORD := BACnetReliability_no_fault_detected;(* ~(BACnet_Reliability 	:		: )	*)
	_PresentValue AT%I*: UDINT; 		(* ~(BACnet_PresentValue 	:		: )
								   			(BACnet_ObjectType 		: MI	: )	*)
	_NumberOfStates AT%I*: UDINT;		(* ~(BACnet_NumberOfStates	:		: )	*)
	_ObjectId AT%I*: DWORD;				(* ~(BACnet_ObjectIdentifier:		: LINK) *)
	_StatusFlags AT%I*: WORD; 			(* ~(BACnet_StatusFlags 	:		: )	*)
	_AckedTransitions AT%I*:WORD;		(* ~(BACnet_AckedTransitions:		: ) *)
	_AckedTransBits : ST_BACnet_EventTransitionBits;
	_nUpdateCount : UDINT := 0;
	_StatusFlagsBits : ST_BACnet_StatusFlags;
END_VAR
(* update server device *)
IF (Device._nUpdateCount = _nUpdateCount) THEN
	Device();
END_IF
(* remind current number of update counter *)
_nUpdateCount := Device._nUpdateCount;

(* handle raw error *)
IF bNoSensor THEN
	_Reliability := BACnetReliability_no_sensor;
ELSIF bOverRange THEN
	_Reliability := BACnetReliability_over_range;
ELSIF bUnderRange THEN
	_Reliability := BACnetReliability_under_range;
ELSIF bOpenLoop THEN
	_Reliability := BACnetReliability_open_loop;
ELSIF bShortedLoop THEN
	_Reliability := BACnetReliability_shorted_loop;
ELSIF bCommFailure THEN
	_Reliability := BACnetReliability_communication_failure;
ELSIF bOtherFault THEN
	_Reliability := BACnetReliability_unreliable_other;
ELSE
	_Reliability := BACnetReliability_no_fault_detected;
END_IF

(* check object type *)
IF (F_BACnet_GetObjType(_ObjectId) <> BACnetObjectType_MultiStateInput) THEN
	(* wrong mapping / invalid object ID *)
	IF _ObjectId = 0 THEN
		nErrorId := BACnet_ERR_WRONG_MAPPING;
	ELSE
		nErrorId := BACnet_ERR_INVALID_OBJECTID;
	END_IF
	bReady := FALSE;

ELSIF (_StatusFlags < 4) OR _AckedTransitions < 5 THEN
	(* wrong mapping *)
	nErrorId := BACnet_ERR_WRONG_MAPPING;
	bReady := FALSE;

ELSIF Device.bOperational THEN
	(* ready state *)
	bReady := TRUE;
	nErrorId := BACnet_ERR_NO_ERROR;

	(* present value *)
	nPresentValue := _PresentValue;

	(* build bit states *)
	_StatusFlagsBits := F_BACnet_StatusFlags(_StatusFlags);
	_AckedTransBits		:= F_BACnet_EventTransitionFlags(_AckedTransitions);

	(* copy states to output *)
	bOverridden := _StatusFlagsBits.overridden;
	bOutOfService := _StatusFlagsBits.out_of_service;
	bFault := _StatusFlagsBits.fault;
	bInAlarm := _StatusFlagsBits.in_alarm;
	bAckedTrans_ToOffNormal := _AckedTransBits.to_offnormal;
	bAckedTrans_ToFault := _AckedTransBits.to_fault;
	bAckedTrans_ToNormal := _AckedTransBits.to_normal;

	(* number of states *)
	nNbrOfStates := _NumberOfStates;

ELSE
	(* server device not ready, reset local ready also *)
	bReady := FALSE;
	nErrorId := BACnet_ERR_OPERATIONAL;
END_IF
(* set error flag *)
bError := (nErrorId <> BACnet_ERR_NO_ERROR);
END_FUNCTION_BLOCK

(* POU FB_BACnet_MultiStateOutput, ST *)
FUNCTION_BLOCK FB_BACnet_MultiStateOutput
VAR_INPUT
	bEnablePV	: BOOL; (* enable present value with priority x in priority array, FALSE = priority x disable *)
	nPV			: UDINT; (* number for priority x, when input bEnablePV is TRUE *)
END_VAR
VAR_IN_OUT
	Device	: FB_BACnet_Device;
END_VAR
VAR_OUTPUT
	bReady			: BOOL;
	nPresentValue	: UDINT;
	bOverridden		: BOOL;
	bOutOfService	: BOOL;
	bFault			: BOOL;
	bInAlarm		: BOOL;
	nNbrOfStates	: UDINT;
	bError			: BOOL;
	nErrorId		: UINT;
END_VAR
VAR
	_PresentValue AT%I*: UDINT; 			(* ~(BACnet_PresentValue 		:		: )
								   				(BACnet_ObjectType			: MO	: )	*)
	_NumberOfStates AT%I*: UDINT;			(* ~(BACnet_NumberOfStates		:		: )	*)
	_StatusFlags AT%I*: WORD; 				(* ~(BACnet_StatusFlags			:		: )	*)
    _PresentValue_Priority12 AT%Q*: UDINT;	(* ~(BACnet_PresentValue_Priority12:	: )	*)
	_StatusFlagsBits : ST_BACnet_StatusFlags;
	_nUpdateCount : UDINT := 0;
END_VAR
(* update server device *)
IF (Device._nUpdateCount = _nUpdateCount) THEN
	Device();
END_IF
(* remind current number of update counter *)
_nUpdateCount := Device._nUpdateCount;

IF Device.bFirstCycle THEN
	(* first call of the server device since reboot/reset *)
	bReady := FALSE;
	_PresentValue_Priority12 := 0;

ELSIF (_StatusFlags < 4) THEN
	(* wrong mapping *)
	nErrorId := BACnet_ERR_WRONG_MAPPING;
	bReady := FALSE;

ELSIF Device.bOperational THEN
	(* ready state *)
	bReady := TRUE;
	nErrorId := BACnet_ERR_NO_ERROR;

	(* write into priority array *)
	IF bEnablePV THEN
		_PresentValue_Priority12	:= nPV;
	ELSE
		_PresentValue_Priority12	:= 0;
	END_IF

	(* present value *)
	nPresentValue := _PresentValue;

	(* build bit states *)
	_StatusFlagsBits := F_BACnet_StatusFlags(_StatusFlags);

	(* copy states to output *)
	bOverridden := _StatusFlagsBits.overridden;
	bOutOfService := _StatusFlagsBits.out_of_service;
	bFault := _StatusFlagsBits.fault;
	bInAlarm := _StatusFlagsBits.in_alarm;

	(* number of states *)
	nNbrOfStates := _NumberOfStates;

ELSE
	(* server device not ready, reset local ready also *)
	bReady := FALSE;
	nErrorId := BACnet_ERR_OPERATIONAL;
END_IF
(* set error flag *)
bError := (nErrorId <> BACnet_ERR_NO_ERROR);
END_FUNCTION_BLOCK

(* POU FB_BACnet_MultiStateOutput_ADS, ST *)
FUNCTION_BLOCK FB_BACnet_MultiStateOutput_ADS
VAR_INPUT
	bEnablePV			: BOOL;
	nPV					: UDINT; (* number for priority x, when input bEnablePV is TRUE *)
	bManual				: BOOL; (* FALSE --> TRUE: write present_value immediately, FALSE: only write present_value on-change, TRUE: write present_value on-change and when device turns operational *)
	ePriority			: E_BACNETPRIORITY := BACNETPRIORITY_12;
END_VAR
VAR_IN_OUT
	Device				: FB_BACnet_Device;
END_VAR
VAR_OUTPUT
	bReady				: BOOL;
	bPvDone				: BOOL; (* present_value written over ADS *)
	nPresentValue		: UDINT;
	bOverridden			: BOOL;
	bOutOfService		: BOOL;
	bFault				: BOOL;
	bInAlarm			: BOOL;
	nNbrOfStates		: UDINT;
	tObjectID			: T_BACnet_ObjectIdentifier := 16#FFFFFFFF;
	bError				: BOOL;
	nErrorId			: UINT;
	nAdsErrorId			: UDINT;
END_VAR
VAR
	_StatusFlags AT%I*: WORD; 				(* ~(BACnet_StatusFlags			:		: )	*)
	_PresentValue AT%I*: UDINT; 			(* ~(BACnet_PresentValue 		:		: )
								   				(BACnet_ObjectType			: MO	: )	*)
	_NumberOfStates AT%I*: UDINT;			(* ~(BACnet_NumberOfStates		:		: )	*)
	_ObjectId AT%I*: DWORD;					(* ~(BACnet_ObjectIdentifier	:		: LINK) *)
	_StatusFlagsBits : ST_BACnet_StatusFlags;
    _PresentValue_Ads : UDINT;
	_nUpdateCount : UDINT := 0;
	_WriteProp : FB_BACnet_WriteProp;
	_rtrigManual : R_TRIG;
	_bEnPvOld : BOOL;
	_nObjType : E_BACNETOBJECTTYPE;
END_VAR
(* update server device *)
IF (Device._nUpdateCount = _nUpdateCount) THEN
	Device();
END_IF
(* remind current number of update counter *)
_nUpdateCount := Device._nUpdateCount;

(* trigger on manual flag *)
_rtrigManual(CLK:= bManual, Q=> );

(* decode object type *)
_nObjType := F_BACnet_GetObjType(_ObjectId);

IF Device.bFirstCycle THEN
	(* first call of the server device since reboot/reset *)
	bReady := FALSE;
	bPvDone := FALSE;

ELSIF _nObjType <> BACnetObjectType_MultiStateOutput THEN
	(* wrong mapped object type *)
	nErrorId := BACnet_ERR_INVALID_OBJECTTYPE;
	bReady := FALSE;
	bPvDone := FALSE;

ELSIF (_StatusFlags < 4) THEN
	(* wrong mapping *)
	nErrorId := BACnet_ERR_WRONG_MAPPING;
	bReady := FALSE;
	bPvDone := FALSE;

ELSIF Device.bOperational THEN

	IF Device.stAdsConn.bValid THEN
		(* write present_value on manual trigger, on-change and on operational recover *)
		IF		_rtrigManual.Q
			OR	((nPV <> _PresentValue_Ads) AND bEnablePV)
			OR	((NOT bReady) AND bManual)
			OR	(bEnablePV <> _bEnPvOld)
		THEN
			_WriteProp.bExecute := TRUE;
			bPvDone := FALSE;
			(* write depending on enable state *)
			IF bEnablePV THEN
				_PresentValue_Ads := nPV;
			ELSE
				_PresentValue_Ads := 0;
			END_IF
			_bEnPvOld := bEnablePV;
		END_IF

		(* ready state *)
		IF (nAdsErrorId = 0) THEN
			bReady := TRUE;
			nErrorId := BACnet_ERR_NO_ERROR;
		END_IF

	ELSE
		(* invalid ADS connection *)
		bReady := FALSE;
		nErrorId := BACnet_ERR_INVALID_ADS_CONN;
		bPvDone := FALSE;
	END_IF

	(* present value *)
	nPresentValue := _PresentValue;

	(* build bit states *)
	_StatusFlagsBits := F_BACnet_StatusFlags(_StatusFlags);

	(* copy states to output *)
	bOverridden := _StatusFlagsBits.overridden;
	bOutOfService := _StatusFlagsBits.out_of_service;
	bFault := _StatusFlagsBits.fault;
	bInAlarm := _StatusFlagsBits.in_alarm;
	tObjectID := _ObjectId;

	(* number of states *)
	nNbrOfStates := _NumberOfStates;

ELSE
	(* server device not ready, reset local ready also *)
	bReady := FALSE;
	nErrorId := BACnet_ERR_OPERATIONAL;
	bPvDone := FALSE;
END_IF

(* call write property command *)
_WriteProp(
	BACnetDevicePort	:= Device.stAdsConn.nAmsPort,
	bExecute			:= ,
	sNetId				:= Device.stAdsConn.sAmsNetId,
	ObjectType			:= _nObjType,
	PropertyID			:= BACnetPropertyIdentifier_PresentValue,
	Priority			:= ePriority,
	DataType			:= BACnetDataType_UnsignedInteger,
	ObjectInstance		:= F_BACnet_GetObjInstance(_ObjectId),
	ptrValue			:= ADR(_PresentValue_Ads),
	nLenValue			:= SIZEOF(_PresentValue_Ads),
	bDone				=> ,
	bBusy				=> ,
	bError				=> ,
	nErrID				=> );

(* set done flag *)
IF _WriteProp.bExecute AND (NOT _WriteProp.bBusy) THEN
	(* check if command was finished with error *)
	IF _WriteProp.bError THEN
		bPvDone		:= FALSE;
		bReady		:= FALSE;
		nErrorId	:= BACnet_ERR_ADS_Write;
	ELSE
		(* successful written *)
		bPvDone		:= TRUE;
	END_IF
	nAdsErrorId := _WriteProp.nErrID;
	(* reset execution bit *)
	_WriteProp(bExecute := FALSE);
END_IF

(* set error flag *)
bError := (nErrorId <> BACnet_ERR_NO_ERROR) OR (nAdsErrorId <> 0);
END_FUNCTION_BLOCK

(* POU FB_BACnet_MultiStateOutput_EX, ST *)
FUNCTION_BLOCK FB_BACnet_MultiStateOutput_EX
VAR_INPUT
	bEnablePV			: BOOL; (* enable present value with priority x in priority array, FALSE = priority x disable *)
	nPV					: UDINT; (* number for priority x, when input bEnablePV is TRUE *)
END_VAR
VAR_IN_OUT
	Device				: FB_BACnet_Device;
END_VAR
VAR_OUTPUT
	bReady				: BOOL;
	nPresentValue		: UDINT;
	bOverridden			: BOOL;
	bOutOfService		: BOOL;
	bFault				: BOOL;
	bInAlarm			: BOOL;
	bNoOutput			: BOOL;
	bOpenLoop			: BOOL;
	bShortedLoop		: BOOL;
	bOtherFault			: BOOL;
	eEventState			: E_BACNETEVENTSTATE;
	bAckedTrans_ToOffNormal : BOOL;
	bAckedTrans_ToFault		: BOOL;
	bAckedTrans_ToNormal	: BOOL;
	nActivePrio			: UINT;
	nNbrOfStates		: UDINT;
	tObjectID			: T_BACnet_ObjectIdentifier := 16#FFFFFFFF;
	bError				: BOOL;
	nErrorId			: UINT;
END_VAR
VAR
	_PresentValue AT%I*: UDINT; 			(* ~(BACnet_PresentValue 		:		: )
								   				(BACnet_ObjectType			: MO	: )	*)
    _PresentValue_Priority12 AT%Q*: UDINT;	(* ~(BACnet_PresentValue_Priority12		:		: )	*)
	_ActivePriority AT%I*: UDINT; 			(* ~(BACnet_ActivePriority 		:		: )	*)
	_NumberOfStates AT%I*: UDINT;			(* ~(BACnet_NumberOfStates		:		: )	*)
	_ObjectId AT%I*: DWORD;					(* ~(BACnet_ObjectIdentifier	:		: LINK) *)
	_StatusFlags AT%I*: WORD; 				(* ~(BACnet_StatusFlags			:		: )	*)
	_EventState AT%I*: WORD;				(* ~(BACnet_EventState			:		: )	*)
	_Reliability AT%I*: WORD; 				(* ~(BACnet_Reliability			:		: )	*)
	_AckedTransitions AT%I*:WORD;			(* ~(BACnet_AckedTransitions	:		: ) *)
	_AckedTransBits : ST_BACnet_EventTransitionBits;
	_nUpdateCount : UDINT := 0;
	_StatusFlagsBits : ST_BACnet_StatusFlags;
END_VAR
(* update server device *)
IF (Device._nUpdateCount = _nUpdateCount) THEN
	Device();
END_IF
(* remind current number of update counter *)
_nUpdateCount := Device._nUpdateCount;

IF Device.bFirstCycle THEN
	(* first call of the server device since reboot/reset *)
	bReady := FALSE;
	_PresentValue_Priority12 := 0;

ELSIF (F_BACnet_GetObjType(_ObjectId) <> BACnetObjectType_MultiStateOutput) THEN
	(* wrong mapping / invalid object ID *)
	IF _ObjectId = 0 THEN
		nErrorId := BACnet_ERR_WRONG_MAPPING;
	ELSE
		nErrorId := BACnet_ERR_INVALID_OBJECTID;
	END_IF
	bReady := FALSE;

ELSIF (_StatusFlags < 4) OR _AckedTransitions < 5 THEN
	(* wrong mapping *)
	nErrorId := BACnet_ERR_WRONG_MAPPING;
	bReady := FALSE;

ELSIF Device.bOperational THEN
	(* ready state *)
	bReady := TRUE;
	nErrorId := BACnet_ERR_NO_ERROR;

	(* write into priority array *)
	IF bEnablePV THEN
		_PresentValue_Priority12	:= nPV;
	ELSE
		_PresentValue_Priority12	:= 0;
	END_IF

	(* present value *)
	nPresentValue := _PresentValue;

	(* build bit states *)
	_StatusFlagsBits := F_BACnet_StatusFlags(_StatusFlags);
	_AckedTransBits		:= F_BACnet_EventTransitionFlags(_AckedTransitions);

	(* copy states to output *)
	bOverridden := _StatusFlagsBits.overridden;
	bOutOfService := _StatusFlagsBits.out_of_service;
	bFault := _StatusFlagsBits.fault;
	bInAlarm := _StatusFlagsBits.in_alarm;
	bNoOutput := (_Reliability = BACnetReliability_no_output);
	bOpenLoop := (_Reliability = BACnetReliability_open_loop);
	bShortedLoop := (_Reliability = BACnetReliability_shorted_loop);
	bOtherFault := (_Reliability = BACnetReliability_unreliable_other);
	bAckedTrans_ToOffNormal := _AckedTransBits.to_offnormal;
	bAckedTrans_ToFault := _AckedTransBits.to_fault;
	bAckedTrans_ToNormal := _AckedTransBits.to_normal;
	tObjectID := _ObjectId;

	(* convert enumeration *)
	eEventState := _EventState;

	(* copy active priority *)
	nActivePrio := UDINT_TO_UINT(_ActivePriority);

	(* number of states *)
	nNbrOfStates := _NumberOfStates;

ELSE
	(* server device not ready, reset local ready also *)
	bReady := FALSE;
	nErrorId := BACnet_ERR_OPERATIONAL;
END_IF
(* set error flag *)
bError := (nErrorId <> BACnet_ERR_NO_ERROR);
END_FUNCTION_BLOCK

(* POU FB_BACnet_MultiStateOutput_RAW, ST *)
FUNCTION_BLOCK FB_BACnet_MultiStateOutput_RAW
VAR_INPUT
	bEnablePV			: BOOL; (* enable present value with priority x in priority array, FALSE = priority x disable *)
	nPV					: UDINT; (* number for priority x, when input bEnablePV is TRUE *)
	nFeedback			AT%Q*: DWORD; (* ~(BACnet_FeedbackValue : : ) *)
	bNoOutput			: BOOL;
	bOpenLoop			: BOOL;
	bShortedLoop		: BOOL;
	bCommFailure		: BOOL;
	bOtherFault			: BOOL;
END_VAR
VAR_IN_OUT
	Device				: FB_BACnet_Device;
END_VAR
VAR_OUTPUT
	bReady				: BOOL;
	nPresentValue		: UDINT;
	bOverridden			: BOOL;
	bOutOfService		: BOOL;
	bFault				: BOOL;
	bInAlarm			: BOOL;
	bAckedTrans_ToOffNormal : BOOL;
	bAckedTrans_ToFault		: BOOL;
	bAckedTrans_ToNormal	: BOOL;
	nNbrOfStates		: UDINT;
	bError				: BOOL;
	nErrorId			: UINT;
	nRawOut				AT%I*: DWORD;		(* ~(BACnet_PresentValue		:		: ) *)
END_VAR
VAR
    _PresentValue_Priority12 AT%Q*: UDINT;	(* ~(BACnet_PresentValue_Priority12:	: )
								   				(BACnet_ObjectType			: MO	: )	*)
	_Reliability AT%Q*: WORD := BACnetReliability_no_fault_detected;(* ~(BACnet_Reliability 	:		: )	*)
	_NumberOfStates AT%I*: UDINT;			(* ~(BACnet_NumberOfStates		:		: )	*)
	_ObjectId AT%I*: DWORD;					(* ~(BACnet_ObjectIdentifier	:		: LINK) *)
	_StatusFlags AT%I*: WORD; 				(* ~(BACnet_StatusFlags			:		: )	*)
	_AckedTransitions AT%I*:WORD;			(* ~(BACnet_AckedTransitions	:		: ) *)
	_AckedTransBits : ST_BACnet_EventTransitionBits;
	_nUpdateCount : UDINT := 0;
	_StatusFlagsBits : ST_BACnet_StatusFlags;
END_VAR
(* update server device *)
IF (Device._nUpdateCount = _nUpdateCount) THEN
	Device();
END_IF
(* remind current number of update counter *)
_nUpdateCount := Device._nUpdateCount;

(* handle raw error *)
IF bNoOutput THEN
	_Reliability := BACnetReliability_no_output;
ELSIF bOpenLoop THEN
	_Reliability := BACnetReliability_open_loop;
ELSIF bShortedLoop THEN
	_Reliability := BACnetReliability_shorted_loop;
ELSIF bCommFailure THEN
	_Reliability := BACnetReliability_communication_failure;
ELSIF bOtherFault THEN
	_Reliability := BACnetReliability_unreliable_other;
ELSE
	_Reliability := BACnetReliability_no_fault_detected;
END_IF

(* check object type *)
IF Device.bFirstCycle THEN
	(* first call of the server device since reboot/reset *)
	bReady := FALSE;
	_PresentValue_Priority12 := 0;

ELSIF (F_BACnet_GetObjType(_ObjectId) <> BACnetObjectType_MultiStateOutput) THEN
	(* wrong mapping / invalid object ID *)
	IF _ObjectId = 0 THEN
		nErrorId := BACnet_ERR_WRONG_MAPPING;
	ELSE
		nErrorId := BACnet_ERR_INVALID_OBJECTID;
	END_IF
	bReady := FALSE;

ELSIF (_StatusFlags < 4) OR _AckedTransitions < 5 THEN
	(* wrong mapping *)
	nErrorId := BACnet_ERR_WRONG_MAPPING;
	bReady := FALSE;

ELSIF Device.bOperational THEN
	(* ready state *)
	bReady := TRUE;
	nErrorId := BACnet_ERR_NO_ERROR;

	(* write into priority array *)
	IF bEnablePV THEN
		_PresentValue_Priority12	:= nPV;
	ELSE
		_PresentValue_Priority12	:= 0;
	END_IF

	(* present value *)
	nPresentValue := nRawOut;

	(* build bit states *)
	_StatusFlagsBits := F_BACnet_StatusFlags(_StatusFlags);
	_AckedTransBits		:= F_BACnet_EventTransitionFlags(_AckedTransitions);

	(* copy states to output *)
	bOverridden := _StatusFlagsBits.overridden;
	bOutOfService := _StatusFlagsBits.out_of_service;
	bFault := _StatusFlagsBits.fault;
	bInAlarm := _StatusFlagsBits.in_alarm;
	bAckedTrans_ToOffNormal := _AckedTransBits.to_offnormal;
	bAckedTrans_ToFault := _AckedTransBits.to_fault;
	bAckedTrans_ToNormal := _AckedTransBits.to_normal;

	(* number of states *)
	nNbrOfStates := _NumberOfStates;

ELSE
	(* server device not ready, reset local ready also *)
	bReady := FALSE;
	nErrorId := BACnet_ERR_OPERATIONAL;
END_IF
(* set error flag *)
bError := (nErrorId <> BACnet_ERR_NO_ERROR);
END_FUNCTION_BLOCK

(* POU FB_BACnet_MultiStateValue, ST *)
FUNCTION_BLOCK FB_BACnet_MultiStateValue
VAR_INPUT
	bEnablePV	: BOOL; (* enable present value with priority x in priority array, FALSE = priority x disable *)
	nPV			: UDINT; (* number for priority x, when input bEnablePV is TRUE *)
END_VAR
VAR_IN_OUT
	Device	: FB_BACnet_Device;
END_VAR
VAR_OUTPUT
	bReady			: BOOL;
	nPresentValue	: UDINT;
	bOverridden		: BOOL;
	bOutOfService	: BOOL;
	bFault			: BOOL;
	bInAlarm		: BOOL;
	nNbrOfStates	: UDINT;
	bError			: BOOL;
	nErrorId		: UINT;
END_VAR
VAR
	_PresentValue AT%I*: UDINT; 			(* ~(BACnet_PresentValue 		:		: )
								   				(BACnet_ObjectType 			: MV	: )	*)
	_NumberOfStates AT%I*: UDINT;			(* ~(BACnet_NumberOfStates		:		: )	*)
	_StatusFlags AT%I*: WORD; 				(* ~(BACnet_StatusFlags 		:		: )	*)
    _PresentValue_Priority12 AT%Q*: UDINT;	(* ~(BACnet_PresentValue_Priority12:	: )	*)
	_nUpdateCount : UDINT := 0;
	_StatusFlagsBits : ST_BACnet_StatusFlags;
END_VAR
(* update server device *)
IF (Device._nUpdateCount = _nUpdateCount) THEN
	Device();
END_IF
(* remind current number of update counter *)
_nUpdateCount := Device._nUpdateCount;

IF Device.bFirstCycle THEN
	(* first call of the server device since reboot/reset *)
	bReady := FALSE;
	_PresentValue_Priority12 := 0;

ELSIF (_StatusFlags < 4) THEN
	(* wrong mapping *)
	nErrorId := BACnet_ERR_WRONG_MAPPING;
	bReady := FALSE;

ELSIF Device.bOperational THEN
	(* ready state *)
	bReady := TRUE;
	nErrorId := BACnet_ERR_NO_ERROR;

	(* write into priority array *)
	IF bEnablePV THEN
		_PresentValue_Priority12	:= nPV;
	ELSE
		_PresentValue_Priority12	:= 0;
	END_IF

	(* present value *)
	nPresentValue := _PresentValue;

	(* build bit states *)
	_StatusFlagsBits := F_BACnet_StatusFlags(_StatusFlags);

	(* copy states to output *)
	bOverridden := _StatusFlagsBits.overridden;
	bOutOfService := _StatusFlagsBits.out_of_service;
	bFault := _StatusFlagsBits.fault;
	bInAlarm := _StatusFlagsBits.in_alarm;

	(* number of states *)
	nNbrOfStates := _NumberOfStates;

ELSE
	(* server device not ready, reset local ready also *)
	bReady := FALSE;
	nErrorId := BACnet_ERR_OPERATIONAL;
END_IF
(* set error flag *)
bError := (nErrorId <> BACnet_ERR_NO_ERROR);
END_FUNCTION_BLOCK

(* POU FB_BACnet_MultiStateValue_ADS, ST *)
FUNCTION_BLOCK FB_BACnet_MultiStateValue_ADS
VAR_INPUT
	bEnablePV			: BOOL;
	nPV					: UDINT; (* number for priority x, when input bEnablePV is TRUE *)
	bManual				: BOOL; (* FALSE --> TRUE: write present_value immediately, FALSE: only write present_value on-change, TRUE: write present_value on-change and when device turns operational *)
	ePriority			: E_BACNETPRIORITY := BACNETPRIORITY_12;
END_VAR
VAR_IN_OUT
	Device				: FB_BACnet_Device;
END_VAR
VAR_OUTPUT
	bReady				: BOOL;
	bPvDone				: BOOL; (* present_value written over ADS *)
	nPresentValue		: UDINT;
	bOverridden			: BOOL;
	bOutOfService		: BOOL;
	bFault				: BOOL;
	bInAlarm			: BOOL;
	nNbrOfStates		: UDINT;
	tObjectID			: T_BACnet_ObjectIdentifier := 16#FFFFFFFF;
	bError				: BOOL;
	nErrorId			: UINT;
	nAdsErrorId			: UDINT;
END_VAR
VAR
	_StatusFlags AT%I*: WORD; 				(* ~(BACnet_StatusFlags 	:		: )	*)
	_PresentValue AT%I*: UDINT; 			(* ~(BACnet_PresentValue 	:		: )
								   				(BACnet_ObjectType 		: MV	: )	*)
	_NumberOfStates AT%I*: UDINT;			(* ~(BACnet_NumberOfStates	:		: )	*)
	_ObjectId AT%I*: DWORD;					(* ~(BACnet_ObjectIdentifier:		: LINK) *)
	_StatusFlagsBits : ST_BACnet_StatusFlags;
    _PresentValue_Ads : UDINT;
	_nUpdateCount : UDINT := 0;
	_WriteProp : FB_BACnet_WriteProp;
	_rtrigManual : R_TRIG;
	_bEnPvOld : BOOL;
	_nObjType : E_BACNETOBJECTTYPE;
END_VAR
(* update server device *)
IF (Device._nUpdateCount = _nUpdateCount) THEN
	Device();
END_IF
(* remind current number of update counter *)
_nUpdateCount := Device._nUpdateCount;

(* trigger on manual flag *)
_rtrigManual(CLK:= bManual, Q=> );

(* decode object type *)
_nObjType := F_BACnet_GetObjType(_ObjectId);

IF Device.bFirstCycle THEN
	(* first call of the server device since reboot/reset *)
	bReady := FALSE;
	bPvDone := FALSE;

ELSIF _nObjType <> BACnetObjectType_MultiStateValue THEN
	(* wrong mapped object type *)
	nErrorId := BACnet_ERR_INVALID_OBJECTTYPE;
	bReady := FALSE;
	bPvDone := FALSE;

ELSIF (_StatusFlags < 4) THEN
	(* wrong mapping *)
	nErrorId := BACnet_ERR_WRONG_MAPPING;
	bReady := FALSE;
	bPvDone := FALSE;

ELSIF Device.bOperational THEN

	IF Device.stAdsConn.bValid THEN
		(* write present_value on manual trigger, on-change and on operational recover *)
		IF		_rtrigManual.Q
			OR	((nPV <> _PresentValue_Ads) AND bEnablePV)
			OR	((NOT bReady) AND bManual)
			OR	(bEnablePV <> _bEnPvOld)
		THEN
			_WriteProp.bExecute := TRUE;
			bPvDone := FALSE;
			(* write depending on enable state *)
			IF bEnablePV THEN
				_PresentValue_Ads := nPV;
			ELSE
				_PresentValue_Ads := 0;
			END_IF
			_bEnPvOld := bEnablePV;
		END_IF

		(* ready state *)
		IF (nAdsErrorId = 0) THEN
			bReady := TRUE;
			nErrorId := BACnet_ERR_NO_ERROR;
		END_IF

	ELSE
		(* invalid ADS connection *)
		bReady := FALSE;
		nErrorId := BACnet_ERR_INVALID_ADS_CONN;
		bPvDone := FALSE;
	END_IF

	(* present value *)
	nPresentValue := _PresentValue;

	(* build bit states *)
	_StatusFlagsBits := F_BACnet_StatusFlags(_StatusFlags);

	(* copy states to output *)
	bOverridden := _StatusFlagsBits.overridden;
	bOutOfService := _StatusFlagsBits.out_of_service;
	bFault := _StatusFlagsBits.fault;
	bInAlarm := _StatusFlagsBits.in_alarm;
	tObjectID := _ObjectId;

	(* number of states *)
	nNbrOfStates := _NumberOfStates;

ELSE
	(* server device not ready, reset local ready also *)
	bReady := FALSE;
	nErrorId := BACnet_ERR_OPERATIONAL;
	bPvDone := FALSE;
END_IF

(* call write property command *)
_WriteProp(
	BACnetDevicePort	:= Device.stAdsConn.nAmsPort,
	bExecute			:= ,
	sNetId				:= Device.stAdsConn.sAmsNetId,
	ObjectType			:= _nObjType,
	PropertyID			:= BACnetPropertyIdentifier_PresentValue,
	Priority			:= ePriority,
	DataType			:= BACnetDataType_UnsignedInteger,
	ObjectInstance		:= F_BACnet_GetObjInstance(_ObjectId),
	ptrValue			:= ADR(_PresentValue_Ads),
	nLenValue			:= SIZEOF(_PresentValue_Ads),
	bDone				=> ,
	bBusy				=> ,
	bError				=> ,
	nErrID				=> );

(* set done flag *)
IF _WriteProp.bExecute AND (NOT _WriteProp.bBusy) THEN
	(* check if command was finished with error *)
	IF _WriteProp.bError THEN
		bPvDone		:= FALSE;
		bReady		:= FALSE;
		nErrorId	:= BACnet_ERR_ADS_Write;
	ELSE
		(* successful written *)
		bPvDone		:= TRUE;
	END_IF
	nAdsErrorId := _WriteProp.nErrID;
	(* reset execution bit *)
	_WriteProp(bExecute := FALSE);
END_IF

(* set error flag *)
bError := (nErrorId <> BACnet_ERR_NO_ERROR) OR (nAdsErrorId <> 0);
END_FUNCTION_BLOCK

(* POU FB_BACnet_MultiStateValue_EX, ST *)
FUNCTION_BLOCK FB_BACnet_MultiStateValue_EX
VAR_INPUT
	bEnablePV			: BOOL; (* enable present value with priority x in priority array, FALSE = priority x disable *)
	nPV					: UDINT; (* number for priority x, when input bEnablePV is TRUE *)
END_VAR
VAR_IN_OUT
	Device				: FB_BACnet_Device;
END_VAR
VAR_OUTPUT
	bReady				: BOOL;
	nPresentValue		: UDINT;
	bOverridden			: BOOL;
	bOutOfService		: BOOL;
	bFault				: BOOL;
	bInAlarm			: BOOL;
	bMultiStateFault	: BOOL;
	bOtherFault			: BOOL;
	eEventState			: E_BACNETEVENTSTATE;
	bAckedTrans_ToOffNormal : BOOL;
	bAckedTrans_ToFault		: BOOL;
	bAckedTrans_ToNormal	: BOOL;
	nActivePrio			: UINT;
	nNbrOfStates		: UDINT;
	tObjectID			: T_BACnet_ObjectIdentifier := 16#FFFFFFFF;
	bError				: BOOL;
	nErrorId			: UINT;
END_VAR
VAR
	_PresentValue AT%I*: UDINT; 			(* ~(BACnet_PresentValue 	:		: )
								   				(BACnet_ObjectType 		: MV	: )	*)
    _PresentValue_Priority12 AT%Q*: UDINT;	(* ~(BACnet_PresentValue_Priority12	:		: )	*)
	_ActivePriority AT%I*: UDINT; 			(* ~(BACnet_ActivePriority 	:		: )	*)
	_NumberOfStates AT%I*: UDINT;			(* ~(BACnet_NumberOfStates	:		: )	*)
	_ObjectId AT%I*: DWORD;					(* ~(BACnet_ObjectIdentifier:		: LINK) *)
	_StatusFlags AT%I*: WORD; 				(* ~(BACnet_StatusFlags 	:		: )	*)
	_EventState AT%I*: WORD;				(* ~(BACnet_EventState 		:		: )	*)
	_Reliability AT%I*: WORD;				(* ~(BACnet_Reliability 	:		: )	*)
	_AckedTransitions AT%I*:WORD;			(* ~(BACnet_AckedTransitions:		: ) *)
	_AckedTransBits : ST_BACnet_EventTransitionBits;
	_StatusFlagsBits : ST_BACnet_StatusFlags;
	_nUpdateCount : UDINT := 0;
END_VAR
(* update server device *)
IF (Device._nUpdateCount = _nUpdateCount) THEN
	Device();
END_IF
(* remind current number of update counter *)
_nUpdateCount := Device._nUpdateCount;

IF Device.bFirstCycle THEN
	(* first call of the server device since reboot/reset *)
	bReady := FALSE;
	_PresentValue_Priority12 := 0;

ELSIF (F_BACnet_GetObjType(_ObjectId) <> BACnetObjectType_MultiStateValue) THEN
	(* wrong mapping / invalid object ID *)
	IF _ObjectId = 0 THEN
		nErrorId := BACnet_ERR_WRONG_MAPPING;
	ELSE
		nErrorId := BACnet_ERR_INVALID_OBJECTID;
	END_IF
	bReady := FALSE;

ELSIF (_StatusFlags < 4) OR _AckedTransitions < 5 THEN
	(* wrong mapping *)
	nErrorId := BACnet_ERR_WRONG_MAPPING;
	bReady := FALSE;

ELSIF Device.bOperational THEN
	(* ready state *)
	bReady := TRUE;
	nErrorId := BACnet_ERR_NO_ERROR;

	(* write into priority array *)
	IF bEnablePV THEN
		_PresentValue_Priority12	:= nPV;
	ELSE
		_PresentValue_Priority12	:= 0;
	END_IF

	(* present value *)
	nPresentValue := _PresentValue;

	(* build bit states *)
	_StatusFlagsBits := F_BACnet_StatusFlags(_StatusFlags);
	_AckedTransBits		:= F_BACnet_EventTransitionFlags(_AckedTransitions);

	(* copy states to output *)
	bOverridden := _StatusFlagsBits.overridden;
	bOutOfService := _StatusFlagsBits.out_of_service;
	bFault := _StatusFlagsBits.fault;
	bInAlarm := _StatusFlagsBits.in_alarm;
	bMultiStateFault := (_Reliability = BACnetReliability_multi_state_fault);
	bOtherFault := (_Reliability = BACnetReliability_unreliable_other);
	bAckedTrans_ToOffNormal := _AckedTransBits.to_offnormal;
	bAckedTrans_ToFault := _AckedTransBits.to_fault;
	bAckedTrans_ToNormal := _AckedTransBits.to_normal;
	tObjectID := _ObjectId;

	(* convert enumeration *)
	eEventState := _EventState;

	(* copy active priority *)
	nActivePrio := UDINT_TO_UINT(_ActivePriority);

	(* number of states *)
	nNbrOfStates := _NumberOfStates;

ELSE
	(* server device not ready, reset local ready also *)
	bReady := FALSE;
	nErrorId := BACnet_ERR_OPERATIONAL;
END_IF
(* set error flag *)
bError := (nErrorId <> BACnet_ERR_NO_ERROR);
END_FUNCTION_BLOCK

(* POU FB_BACnet_NotificationClass, ST *)
FUNCTION_BLOCK FB_BACnet_NotificationClass
VAR_IN_OUT
	Device	: FB_BACnet_Device;
END_VAR
VAR_OUTPUT
	bReady			: BOOL;
	bError			: BOOL;
	nErrorId		: UINT;
END_VAR
VAR
	_ObjectId AT%I* : DWORD;					(* ~(BACnet_ObjectIdentifier:		: LINK)
													(BACnet_ObjectType		:	NC	: ) *)
	_nUpdateCount	: UDINT := 0;
END_VAR
(* update server device *)
IF (Device._nUpdateCount = _nUpdateCount) THEN
	Device();
END_IF
(* remind current number of update counter *)
_nUpdateCount := Device._nUpdateCount;

IF Device.bOperational THEN
	(* ready state *)
	bReady := TRUE;
	nErrorId := BACnet_ERR_NO_ERROR;
ELSE
	(* server device not ready, reset local ready also *)
	bReady := FALSE;
	nErrorId := BACnet_ERR_OPERATIONAL;
END_IF
(* set error flag *)
bError := (nErrorId <> BACnet_ERR_NO_ERROR);
END_FUNCTION_BLOCK

(* POU FB_BACnet_NotificationClass_EX, ST *)
FUNCTION_BLOCK FB_BACnet_NotificationClass_EX
VAR_IN_OUT
	Device				: FB_BACnet_Device;
END_VAR
VAR_OUTPUT
	bReady				: BOOL;
	tObjectID			: T_BACnet_ObjectIdentifier := 16#FFFFFFFF;
	bError				: BOOL;
	nErrorId			: UINT;
END_VAR
VAR
	_ObjectId AT%I* : DWORD;					(* ~(BACnet_ObjectIdentifier:		: LINK)
													(BACnet_ObjectType		:	NC	: ) *)
	_nUpdateCount	: UDINT := 0;
END_VAR
(* update server device *)
IF (Device._nUpdateCount = _nUpdateCount) THEN
	Device();
END_IF
(* remind current number of update counter *)
_nUpdateCount := Device._nUpdateCount;

IF (F_BACnet_GetObjType(_ObjectId) <> BACnetObjectType_NotificationClass) THEN
	(* wrong mapping / invalid object ID *)
	IF _ObjectId = 0 THEN
		nErrorId := BACnet_ERR_WRONG_MAPPING;
	ELSE
		nErrorId := BACnet_ERR_INVALID_OBJECTID;
	END_IF
	bReady := FALSE;
	tObjectID := 16#FFFFFFFF;

ELSIF Device.bOperational THEN
	(* ready state *)
	bReady := TRUE;
	nErrorId := BACnet_ERR_NO_ERROR;
	tObjectID := _ObjectId;

ELSE
	(* server device not ready, reset local ready also *)
	bReady := FALSE;
	nErrorId := BACnet_ERR_OPERATIONAL;
END_IF
(* set error flag *)
bError := (nErrorId <> BACnet_ERR_NO_ERROR);
END_FUNCTION_BLOCK

(* POU FB_BACnet_NotificationSinkDelEntry, ST *)
FUNCTION_BLOCK FB_BACnet_NotificationSinkDelEntry
VAR_INPUT
	bExecute	: BOOL;
	nIndex		: UDINT;
	sNetId		: T_AmsNetId;
	nPort		: T_AmsPort;
	tTimeout	: TIME := BACnet_ADSTimeOut;
END_VAR
VAR_OUTPUT
	bBusy		: BOOL;
	bEmpty		: BOOL;
	bError		: BOOL;
	nErrorId	: UDINT;
END_VAR
VAR
	_AdsReadClient	: ADSREAD;
END_VAR
	_AdsReadClient(
		NETID	:= sNetId,
		PORT	:= nPort,
		IDXGRP	:= 16#5,
		IDXOFFS	:= nIndex,
		LEN		:= 0,
		DESTADDR:= 0,
		READ	:= bExecute,
		TMOUT	:= tTimeout,
		BUSY	=> bBusy,
		ERR		=> bError,
		ERRID	=> nErrorId);

	bEmpty := ((UDINT_TO_DWORD(_AdsReadClient.ERRID) AND 16#FFF) = 16#703);
END_FUNCTION_BLOCK

(* POU FB_BACnet_ObjectListProperty, ST *)
FUNCTION_BLOCK FB_BACnet_ObjectListProperty
VAR_INPUT
	bAutoGet			: BOOL:=TRUE; (* TRUE = get data from property when ADS connection OR object ID changed *)
	bGet				: BOOL; (* FALSE --> TRUE = get data from property *)
	bTypeFilter			: BOOL; (* activate input "eObjectTypeFilter" *)
	eObjType			: E_BACnetObjectType; (* select the object type that is scanned *)
END_VAR
VAR_IN_OUT
	stAdsConn			: ST_BACnet_AdsConnection;
END_VAR
VAR_OUTPUT
	bDone				: BOOL;
	bBusy				: BOOL;
	bError				: BOOL;
	nErrorId			: UINT;
	stObjIDList			: ST_BACnet_ObjectIdentifierList;
END_VAR
VAR
	_fbReadProp			: FB_BACnet_ReadProp;
	_i					: INT;
	_cbPropSize			: UDINT;
	_cbMemCpy			: UDINT;
	_nEntryCount		: UDINT;
	_iScan				: UDINT;
	_pEntry				: POINTER TO T_BACnet_ObjectIdentifier := 16#FFFFFFFF;
	_cbAdsBuf			: UDINT;
	_rtrigGetSet		: R_TRIG;
	_nAdsReloadOld		: USINT;
	_bUseObjTypeFilterOld: BOOL;
	_eObjTypeFilterOld	: E_BACnetObjectType;
	_nDeviceIdOld		: DWORD := 16#FFFFFFFF;
END_VAR
(* ADS read *);
_fbReadProp(
	BACnetDevicePort	:= stAdsConn.nAmsPort,
	bExecute			:= ,
	ObjectInstance		:= F_BACnet_GetObjInstance(stAdsConn.nDeviceId),
	ObjectType			:= BACnetObjectType_Device,
	sNetId				:= stAdsConn.sAmsNetId,
	PropertyID			:= BACnetPropertyIdentifier_ObjectList,
	DataType			:= BACnetDataType_ObjectIdentifierArr,
	ptrValue			:= ADR(stBACnet_AdsBuffer.arrData),
	nLenValue			:= SIZEOF(stBACnet_AdsBuffer.arrData),
	bDone				=> ,
	bBusy				=> ,
	bError				=> ,
	nErrID				=> ,
	nProcessedLen		=> );

(* trigger start event *)
_rtrigGetSet(CLK:= bGet, Q=> );

(* state machine *)
CASE _i OF

	0: (* Idle *)
		IF		(		(
								(_nAdsReloadOld <> stAdsConn.nReload)
							OR	(_bUseObjTypeFilterOld <> bTypeFilter)
							OR	((_eObjTypeFilterOld <> eObjType) AND bTypeFilter)
							OR	(_nDeviceIdOld <> stAdsConn.nDeviceId)
						)
					AND	bAutoGet
				)
			OR	_rtrigGetSet.Q
		THEN
			IF (NOT stAdsConn.bValid) THEN
				(* ADS connection not valid *)
				nErrorId := BACnet_ERR_INVALID_ADS_CONN;
			ELSE
				nErrorId := BACnet_ERR_NO_ERROR;
				_i := 1;
				(* remind ADS reload counter and parameter *)
				_nAdsReloadOld := stAdsConn.nReload;
				_bUseObjTypeFilterOld := bTypeFilter;
				_eObjTypeFilterOld := eObjType;
				_nDeviceIdOld := stAdsConn.nDeviceId;
			END_IF
			(* reset done flag *)
			bDone := FALSE;
		END_IF
		IF (NOT bGet) AND (NOT bAutoGet) THEN
			nErrorId := BACnet_ERR_NO_ERROR;
			bDone := FALSE;
		END_IF

	(* READ *)
	1: (* read object property data via ADS *)
		IF TestAndSet(stBACnet_AdsBuffer.bTestSet) THEN
			IF _fbReadProp.bExecute THEN
				IF _fbReadProp.bError THEN
					_i := 100;
					nErrorId := BACnet_ERR_ADS_Read;
					_fbReadProp.bExecute := FALSE;
				ELSIF (NOT _fbReadProp.bBusy) THEN
					_fbReadProp.bExecute := FALSE;
					_cbPropSize := _fbReadProp.nProcessedLen;
					(* clear output data *)
					MEMSET(ADR(stObjIDList), 0, SIZEOF(stObjIDList));
					(* check if the ADS buffer reached its ending *)
					IF _cbPropSize > _cbAdsBuf THEN
						(* ADS buffer too small *)
						nErrorId := BACnet_ERR_ADS_BufferSize;
						(* reduce size of data to copy *)
						IF (_cbAdsBuf MOD 4) <> 0 THEN
							_cbPropSize := _F_BACnet_AlignedSize(_cbAdsBuf - 4);
						ELSE
							_cbPropSize := _cbAdsBuf;
						END_IF
					END_IF

					(* filter object type or not? *)
					IF NOT bTypeFilter THEN
						(* copy all from ADS buffer *)
						_cbMemCpy := MEMCPY(	ADR(stObjIDList.arrObjList),
												ADR(stBACnet_AdsBuffer.arrData),
												MIN(_cbPropSize, SIZEOF(stObjIDList.arrObjList))
						);
						IF _cbMemCpy < _cbPropSize THEN
							(* not all property data copied *)
							nErrorId := BACnet_ERR_ADS_TooManyObjects;
						END_IF
						(* how many entries read? *)
						stObjIDList.nEntries := _cbMemCpy / 4;
					ELSE
						(* filter - scan entry by entry *)
						_nEntryCount := _cbPropSize / 4;
						_iScan := 0;
						_pEntry := ADR(stBACnet_AdsBuffer.arrData);
						_cbPropSize := _pEntry + _cbPropSize;
						(* scan entry by entry and add to list if matching with filter *)
						WHILE (		(_pEntry + 4) <= _cbPropSize)
								AND	(_iScan < _nEntryCount)
						DO
							IF F_BACnet_GetObjType(_pEntry^) = eObjType THEN
								(* add item to list *)
								stObjIDList.arrObjList[stObjIDList.nEntries] := _pEntry^;
								stObjIDList.nEntries := stObjIDList.nEntries + 1;
							END_IF
							(* count up *)
							_iScan := _iScan + 1;
							_pEntry := _pEntry + SIZEOF(_pEntry^);
						END_WHILE
					END_IF
					(* DONE *)
					_i := 100;
				END_IF

			ELSIF (stBACnet_AdsBuffer.iLocked = 0) THEN
				_fbReadProp.bExecute := TRUE;
				(* lock global ADS buffer *)
				_cbAdsBuf := SIZEOF(stBACnet_AdsBuffer.arrData);
				stBACnet_AdsBuffer.iLocked := _cbAdsBuf;
			END_IF

			(* release temporary task lock *)
			stBACnet_AdsBuffer.bTestSet := FALSE;
		END_IF

	100: (* Done *)
		bDone := (nErrorId = BACnet_ERR_NO_ERROR);
		(* release ADS buffer *)
		stBACnet_AdsBuffer.iLocked := 0;
		_i := 0;

END_CASE

(* set error flag *)
bError 	:= nErrorId > BACnet_ERR_NO_ERROR;
bBusy 	:= _i > 0;
END_FUNCTION_BLOCK

(* POU FB_BACnet_Program, ST *)
FUNCTION_BLOCK FB_BACnet_Program
VAR_INPUT
	bRelease			: BOOL;
	bCommonError		: BOOL;
	bWaitForSomething	: BOOL;
	stDoneFlags			: ST_BACnet_ProgramHandshakeRequests;
	stFailedFlags		: ST_BACnet_ProgramHandshakeRequests;
	bModeUnloadComplex	: BOOL := TRUE;
END_VAR
VAR_IN_OUT
	Device				: FB_BACnet_Device;
END_VAR
VAR_OUTPUT
	bReady				: BOOL;
	bOverridden			: BOOL;
	bOutOfService		: BOOL;
	bFault				: BOOL;
	bInAlarm			: BOOL;
	stRequestFlags		: ST_BACnet_ProgramHandshakeRequests;
	stActiveStateFlags	: ST_BACnet_ProgramHandshakeStates;
	bError				: BOOL;
	nErrorId			: UINT;
END_VAR
VAR
(* from BACnet to PLC *)
	_ProgramChange AT%I*: WORD;			(* ~(BACnet_ProgramChange 				:		: )
											(BACnet_ObjectType 					: PROG	: ) *)
	_StatusFlags AT%I*: WORD;			(* ~(BACnet_StatusFlags 				:		: )	*)

(* from PLC to BACnet *)
	_ProgramState AT%Q*: WORD;			(* ~(BACnet_ProgramState 				:		: ) *)
	_ReasonForHalt AT%Q*: WORD;			(* ~(BACnet_ReasonForHalt 				:		: )	*)
	_SetProgramReadyState AT%Q*: BOOL;	(* ~(BACnet_SetProgramReadyState 		:		: )	*)

(* internal signals *)
	_StatusFlagsBits 	: ST_BACnet_StatusFlags;
	_bTriggerSetup		: BOOL;
	_ActiveChange		: E_BACNETPROGRAMREQUEST; (* ACTIVE PROGRAM CHANGE *)
	_bLockedForChange	: BOOL;
	_nUpdateCount		: UDINT := 0;
END_VAR
(* update server device *)
IF (Device._nUpdateCount = _nUpdateCount) THEN
	Device();
END_IF
(* remind current number of update counter *)
_nUpdateCount := Device._nUpdateCount;

(* check BitString format of StatusFlags --> if StatusFlags are less than 4, object isn't linked correctly *)
IF (_StatusFlags < 4) THEN
	(* wrong mapping *)
	nErrorId := BACnet_ERR_WRONG_MAPPING;
	bReady := FALSE;

ELSIF Device.bOperational THEN
	(* ready state *)
	bReady := TRUE;
	nErrorId := BACnet_ERR_NO_ERROR;

	(* decode status flags *)
	_StatusFlagsBits := F_BACnet_StatusFlags(_StatusFlags);

	(* copy states to output *)
	bOverridden := _StatusFlagsBits.overridden;
	bOutOfService := _StatusFlagsBits.out_of_service;
	bFault := _StatusFlagsBits.fault;
	bInAlarm := _StatusFlagsBits.in_alarm;

	(* execute change *)
	CASE _ActiveChange OF
		BACnetProgramRequest_ready:
			(* idle *);

		BACnetProgramRequest_load:
			_ProgramState	:= BACnetProgramState_loading;
			_ActiveChange	:= BACnetProgramRequest_ready;

		BACnetProgramRequest_restart,
		BACnetProgramRequest_run:
			IF _bTriggerSetup THEN
				(* wait on setup finish *)
				IF stFailedFlags.bSetup OR bCommonError OR (NOT bRelease) THEN
					(* abort *)
					_ProgramState := BACnetProgramState_halted;
					_ActiveChange := BACnetProgramRequest_ready;
					_ReasonForHalt := BACnetProgramError_progerror_internal;
				ELSIF stDoneFlags.bSetup THEN
					(* setup done, start "normal" running mode *)
					_bTriggerSetup := FALSE;
					_ActiveChange := BACnetProgramRequest_run;
				END_IF
			ELSE
				IF stFailedFlags.bRun OR bCommonError OR (NOT bRelease) THEN
					(* abort *)
					_ProgramState := BACnetProgramState_halted;
					_ActiveChange := BACnetProgramRequest_ready;
					_ReasonForHalt := BACnetProgramError_progerror_internal;
				ELSIF stDoneFlags.bRun THEN
					(* switch to running state *)
					_ProgramState := BACnetProgramState_running;
					_ActiveChange := BACnetProgramRequest_ready;
				END_IF
			END_IF

		BACnetProgramRequest_halt:
			(* wait on halted *)
			IF stFailedFlags.bHalt OR bCommonError OR (NOT bRelease) THEN
				(* abort *)
				_ProgramState := BACnetProgramState_halted;
				_ActiveChange := BACnetProgramRequest_ready;
				_ReasonForHalt := BACnetProgramError_progerror_internal;
			ELSIF stDoneFlags.bHalt THEN
				(* halted *)
				_ProgramState := BACnetProgramState_halted;
				_ActiveChange := BACnetProgramRequest_ready;
				_ReasonForHalt := BACnetProgramError_program;
			END_IF

		BACnetProgramRequest_unload:
			_ProgramState	:= BACnetProgramState_unloading;
			_ActiveChange	:= BACnetProgramRequest_ready;

	END_CASE

	(* start change request and handle error states *)
	IF (_ActiveChange = BACnetProgramRequest_ready) THEN

		CASE _ProgramState OF
			BACnetProgramState_idle:
				IF bCommonError THEN
					(* abort *)
					_ProgramState := BACnetProgramState_halted;
					_ReasonForHalt := BACnetProgramError_progerror_internal;
				ELSIF (NOT bRelease) THEN
					(* abort *)
					_ProgramState := BACnetProgramState_halted;
					_ReasonForHalt := BACnetProgramError_other;
				ELSIF (NOT _bLockedForChange) THEN
					_ReasonForHalt := BACnetProgramError_program_normal;
					CASE _ProgramChange OF
						BACnetProgramRequest_unload,
						BACnetProgramRequest_halt:
							(* acknowledge without execution *)
							_SetProgramReadyState	:= TRUE;
						BACnetProgramRequest_restart,
						BACnetProgramRequest_run,
						BACnetProgramRequest_load:
							(* execute request *)
							_ActiveChange := BACnetProgramRequest_load;
							_bTriggerSetup := TRUE;
					END_CASE
				END_IF

			BACnetProgramState_loading:
				IF bCommonError THEN
					(* abort *)
					_ProgramState := BACnetProgramState_halted;
					_ReasonForHalt := BACnetProgramError_progerror_internal;
				ELSIF (NOT bRelease) THEN
					(* abort *)
					_ProgramState := BACnetProgramState_halted;
					_ReasonForHalt := BACnetProgramError_other;
				ELSIF stFailedFlags.bLoad THEN
					(* abort *)
					_ProgramState := BACnetProgramState_halted;
					_ReasonForHalt := BACnetProgramError_load_failed;
				ELSIF stDoneFlags.bLoad THEN
					(* DONE *)
					_bTriggerSetup := TRUE;
					_ActiveChange := BACnetProgramRequest_run;
				ELSIF (NOT _bLockedForChange) THEN
					_ReasonForHalt := BACnetProgramError_program_normal;
					CASE _ProgramChange OF
						BACnetProgramRequest_load,
						BACnetProgramRequest_run,
						BACnetProgramRequest_halt,
						BACnetProgramRequest_restart:
							(* acknowledge without execution *)
							_SetProgramReadyState	:= TRUE;
						BACnetProgramRequest_unload:
							(* execute request *)
							_ActiveChange := _ProgramChange;
					END_CASE
				END_IF

			BACnetProgramState_running:
				IF bCommonError THEN
					(* abort *)
					_ProgramState := BACnetProgramState_halted;
					_ReasonForHalt := BACnetProgramError_progerror_internal;
				ELSIF (NOT bRelease) THEN
					(* abort *)
					_ProgramState := BACnetProgramState_halted;
					_ReasonForHalt := BACnetProgramError_other;
				ELSIF bWaitForSomething THEN
					(* wait on something *)
					_ProgramState := BACnetProgramState_waiting;
				ELSIF (NOT _bLockedForChange) THEN
					_ReasonForHalt := BACnetProgramError_program_normal;
					CASE _ProgramChange OF
						BACnetProgramRequest_run:
							(* is already running *)
							_SetProgramReadyState	:= TRUE;
						BACnetProgramRequest_unload,
						BACnetProgramRequest_halt:
							(* execute request *)
							_ActiveChange := _ProgramChange;
						BACnetProgramRequest_restart,
						BACnetProgramRequest_load:
							(* retrigger setup *)
							_ActiveChange := BACnetProgramRequest_restart;
							_bTriggerSetup := TRUE;
					END_CASE
				END_IF

			BACnetProgramState_waiting:
				IF bCommonError THEN
					(* abort *)
					_ProgramState := BACnetProgramState_halted;
					_ReasonForHalt := BACnetProgramError_progerror_internal;
				ELSIF (NOT bRelease) THEN
					(* abort *)
					_ProgramState := BACnetProgramState_halted;
					_ReasonForHalt := BACnetProgramError_other;
				ELSIF (NOT bWaitForSomething) THEN
					(* got it *)
					_ProgramState := BACnetProgramState_running;
				ELSIF (NOT _bLockedForChange) THEN
					_ReasonForHalt := BACnetProgramError_program_normal;
					CASE _ProgramChange OF
						BACnetProgramRequest_run:
							(* is already running *)
							_SetProgramReadyState	:= TRUE;
						BACnetProgramRequest_unload,
						BACnetProgramRequest_halt:
							(* execute request *)
							_ActiveChange := _ProgramChange;
					END_CASE
				END_IF

			BACnetProgramState_halted:
				IF (NOT bCommonError) AND bRelease AND (NOT _bLockedForChange) THEN
					CASE _ProgramChange OF
						BACnetProgramRequest_halt:
							(* acknowledge without execution *)
							_SetProgramReadyState	:= TRUE;
						BACnetProgramRequest_unload:
							(* execute request *)
							_ActiveChange := _ProgramChange;
						BACnetProgramRequest_restart,
						BACnetProgramRequest_load:
							(* retrigger setup *)
							_ActiveChange := BACnetProgramRequest_restart;
							_bTriggerSetup := TRUE;
						BACnetProgramRequest_run:
							(* start, but don't trigger setup *)
							_ActiveChange := _ProgramChange;
							_bTriggerSetup := FALSE;
					END_CASE
				END_IF

			BACnetProgramState_unloading:
				IF bModeUnloadComplex THEN
					_ReasonForHalt := BACnetProgramError_program_normal;
					IF bCommonError THEN
						(* abort *)
						_ProgramState := BACnetProgramState_halted;
						_ActiveChange := BACnetProgramRequest_ready;
						_ReasonForHalt := BACnetProgramError_progerror_internal;
					ELSIF (NOT bRelease) THEN
						(* abort *)
						_ProgramState := BACnetProgramState_halted;
						_ActiveChange := BACnetProgramRequest_ready;
						_ReasonForHalt := BACnetProgramError_other;
					ELSIF stFailedFlags.bUnload THEN
						(* abort *)
						_ProgramState := BACnetProgramState_halted;
						_ActiveChange := BACnetProgramRequest_ready;
						_ReasonForHalt := BACnetProgramError_other;
					ELSIF stDoneFlags.bUnload THEN
						(* DONE *)
						_ActiveChange := BACnetProgramRequest_ready;
						_ProgramState := BACnetProgramState_idle;
					ELSIF (NOT _bLockedForChange) THEN
						CASE _ProgramChange OF
							BACnetProgramRequest_load,
							BACnetProgramRequest_run,
							BACnetProgramRequest_halt,
							BACnetProgramRequest_restart,
							BACnetProgramRequest_unload:
								(* acknowledge without execution *)
								_SetProgramReadyState	:= TRUE;
						END_CASE
					END_IF
				END_IF

		END_CASE
	END_IF

	(* check state of "change" request *)
	IF (_ActiveChange <> BACnetProgramRequest_ready) THEN
		(* request is active, lock execution *)
		_bLockedForChange		:= TRUE;
	ELSIF _bLockedForChange AND (NOT _SetProgramReadyState) THEN
		(* change finished, tell the stack done *)
		_SetProgramReadyState	:= TRUE;
		_bTriggerSetup			:= FALSE;
	ELSIF (_ProgramChange = BACnetProgramRequest_ready) THEN
		(* wait on new requests *)
		_SetProgramReadyState	:= FALSE;
		_bLockedForChange		:= FALSE;
		_bTriggerSetup			:= FALSE;
	ELSE
		(* new request *)
		_bTriggerSetup			:= FALSE;
	END_IF

	(* external requests *)
	stRequestFlags.bLoad			:= (_ProgramState = BACnetProgramState_loading) AND (NOT _bLockedForChange);
	stRequestFlags.bSetup			:=	(		(_ActiveChange = BACnetProgramRequest_run)
										OR	(_ActiveChange = BACnetProgramRequest_restart)
									)
								AND	_bTriggerSetup;
	stRequestFlags.bRun			:= (_ActiveChange = BACnetProgramRequest_run) AND (NOT _bTriggerSetup);
	stRequestFlags.bHalt			:= _ActiveChange = BACnetProgramRequest_halt;
	stRequestFlags.bUnload		:=	(_ActiveChange = BACnetProgramRequest_unload)
								OR	(		(_ProgramState = BACnetProgramState_unloading)
										AND	(NOT _bLockedForChange)
									);

	(* active status flags *)
	stActiveStateFlags.bIdle		:= _ProgramState = BACnetProgramState_idle;
	stActiveStateFlags.bLoading		:= _ProgramState = BACnetProgramState_loading;
	stActiveStateFlags.bRunning		:= _ProgramState = BACnetProgramState_running;
	stActiveStateFlags.bWaiting		:= _ProgramState = BACnetProgramState_waiting;
	stActiveStateFlags.bHalted		:= _ProgramState = BACnetProgramState_halted;
	stActiveStateFlags.bUnloading	:= _ProgramState = BACnetProgramState_unloading;
ELSE
	(* server device not ready, reset local ready also *)
	bReady := FALSE;
	nErrorId := BACnet_ERR_OPERATIONAL;
END_IF
(* set error flag *)
bError := (nErrorId <> BACnet_ERR_NO_ERROR);
END_FUNCTION_BLOCK

(* POU FB_BACnet_Program_EX, ST *)
FUNCTION_BLOCK FB_BACnet_Program_EX
VAR_INPUT
	bRelease			: BOOL;
	bCommonError		: BOOL;
	bWaitForSomething	: BOOL;
	stDoneFlags			: ST_BACnet_ProgramHandshakeRequests;
	stFailedFlags		: ST_BACnet_ProgramHandshakeRequests;
	bModeUnloadComplex	: BOOL := TRUE;
END_VAR
VAR_IN_OUT
	Device				: FB_BACnet_Device;
END_VAR
VAR_OUTPUT
	bReady				: BOOL;
	bOverridden			: BOOL;
	bOutOfService		: BOOL;
	bFault				: BOOL;
	bInAlarm			: BOOL;
	bProcessError		: BOOL;
	bCommFailure		: BOOL;
	bOtherFault			: BOOL;
	stRequestFlags		: ST_BACnet_ProgramHandshakeRequests;
	stActiveStateFlags	: ST_BACnet_ProgramHandshakeStates;
	tObjectID			: T_BACnet_ObjectIdentifier := 16#FFFFFFFF;
	bError				: BOOL;
	nErrorId			: UINT;
END_VAR
VAR
(* from BACnet to PLC *)
	_ObjectId AT%I* : DWORD;			(* ~(BACnet_ObjectIdentifier	:		: LINK) *)
	_ProgramChange AT%I*: WORD;			(* ~(BACnet_ProgramChange 		:		: )
											(BACnet_ObjectType 			: PROG	: ) *)
	_StatusFlags AT%I*: WORD;			(* ~(BACnet_StatusFlags 		:		: )	*)
	_Reliability AT%I*: WORD;			(* ~(BACnet_Reliability 		:		: )	*)

(* from PLC to BACnet *)
	_ProgramState AT%Q*: WORD;			(* ~(BACnet_ProgramState 		:		: ) *)
	_ReasonForHalt AT%Q*: WORD;			(* ~(BACnet_ReasonForHalt 		:		: )	*)
	_SetProgramReadyState AT%Q*: BOOL;	(* ~(BACnet_SetProgramReadyState:		: )	*)

(* internal signals *)
	_StatusFlagsBits 	: ST_BACnet_StatusFlags;
	_bTriggerSetup		: BOOL;
	_ActiveChange		: E_BACNETPROGRAMREQUEST; (* ACTIVE PROGRAM CHANGE *)
	_bLockedForChange	: BOOL;
	_nUpdateCount		: UDINT := 0;
END_VAR
(* update server device *)
IF (Device._nUpdateCount = _nUpdateCount) THEN
	Device();
END_IF
(* remind current number of update counter *)
_nUpdateCount := Device._nUpdateCount;

(* check BitString format of StatusFlags --> if StatusFlags are less than 4, object isn't linked correctly *)
IF (F_BACnet_GetObjType(_ObjectId) <> BACnetObjectType_Program) THEN
	(* wrong mapping / invalid object ID *)
	IF _ObjectId = 0 THEN
		nErrorId := BACnet_ERR_WRONG_MAPPING;
	ELSE
		nErrorId := BACnet_ERR_INVALID_OBJECTID;
	END_IF
	bReady := FALSE;
	tObjectID := 16#FFFFFFFF;

ELSIF (_StatusFlags < 4) THEN
	(* wrong mapping *)
	nErrorId := BACnet_ERR_WRONG_MAPPING;
	bReady := FALSE;

ELSIF Device.bOperational THEN
	(* ready state *)
	bReady := TRUE;
	nErrorId := BACnet_ERR_NO_ERROR;

	(* decode status flags *)
	_StatusFlagsBits := F_BACnet_StatusFlags(_StatusFlags);

	(* copy states to output *)
	bOverridden := _StatusFlagsBits.overridden;
	bOutOfService := _StatusFlagsBits.out_of_service;
	bFault := _StatusFlagsBits.fault;
	bInAlarm := _StatusFlagsBits.in_alarm;
	bProcessError := (_Reliability = BACnetReliability_process_error);
	bCommFailure := (_Reliability = BACnetReliability_communication_failure);
	bOtherFault := (_Reliability = BACnetReliability_unreliable_other);
	tObjectID := _ObjectId;

	(* execute change *)
	CASE _ActiveChange OF
		BACnetProgramRequest_ready:
			(* idle *);

		BACnetProgramRequest_load:
			_ProgramState	:= BACnetProgramState_loading;
			_ActiveChange	:= BACnetProgramRequest_ready;

		BACnetProgramRequest_restart,
		BACnetProgramRequest_run:
			IF _bTriggerSetup THEN
				(* wait on setup finish *)
				IF stFailedFlags.bSetup OR bCommonError OR (NOT bRelease) THEN
					(* abort *)
					_ProgramState := BACnetProgramState_halted;
					_ActiveChange := BACnetProgramRequest_ready;
					_ReasonForHalt := BACnetProgramError_progerror_internal;
				ELSIF stDoneFlags.bSetup THEN
					(* setup done, start "normal" running mode *)
					_bTriggerSetup := FALSE;
					_ActiveChange := BACnetProgramRequest_run;
				END_IF
			ELSE
				IF stFailedFlags.bRun OR bCommonError OR (NOT bRelease) THEN
					(* abort *)
					_ProgramState := BACnetProgramState_halted;
					_ActiveChange := BACnetProgramRequest_ready;
					_ReasonForHalt := BACnetProgramError_progerror_internal;
				ELSIF stDoneFlags.bRun THEN
					(* switch to running state *)
					_ProgramState := BACnetProgramState_running;
					_ActiveChange := BACnetProgramRequest_ready;
				END_IF
			END_IF

		BACnetProgramRequest_halt:
			(* wait on halted *)
			IF stFailedFlags.bHalt OR bCommonError OR (NOT bRelease) THEN
				(* abort *)
				_ProgramState := BACnetProgramState_halted;
				_ActiveChange := BACnetProgramRequest_ready;
				_ReasonForHalt := BACnetProgramError_progerror_internal;
			ELSIF stDoneFlags.bHalt THEN
				(* halted *)
				_ProgramState := BACnetProgramState_halted;
				_ActiveChange := BACnetProgramRequest_ready;
				_ReasonForHalt := BACnetProgramError_program;
			END_IF

		BACnetProgramRequest_unload:
			_ProgramState	:= BACnetProgramState_unloading;
			_ActiveChange	:= BACnetProgramRequest_ready;

	END_CASE

	(* start change request and handle error states *)
	IF (_ActiveChange = BACnetProgramRequest_ready) THEN

		CASE _ProgramState OF
			BACnetProgramState_idle:
				IF bCommonError THEN
					(* abort *)
					_ProgramState := BACnetProgramState_halted;
					_ReasonForHalt := BACnetProgramError_progerror_internal;
				ELSIF (NOT bRelease) THEN
					(* abort *)
					_ProgramState := BACnetProgramState_halted;
					_ReasonForHalt := BACnetProgramError_other;
				ELSIF (NOT _bLockedForChange) THEN
					_ReasonForHalt := BACnetProgramError_program_normal;
					CASE _ProgramChange OF
						BACnetProgramRequest_unload,
						BACnetProgramRequest_halt:
							(* acknowledge without execution *)
							_SetProgramReadyState	:= TRUE;
						BACnetProgramRequest_restart,
						BACnetProgramRequest_run,
						BACnetProgramRequest_load:
							(* execute request *)
							_ActiveChange := BACnetProgramRequest_load;
							_bTriggerSetup := TRUE;
					END_CASE
				END_IF

			BACnetProgramState_loading:
				IF bCommonError THEN
					(* abort *)
					_ProgramState := BACnetProgramState_halted;
					_ReasonForHalt := BACnetProgramError_progerror_internal;
				ELSIF (NOT bRelease) THEN
					(* abort *)
					_ProgramState := BACnetProgramState_halted;
					_ReasonForHalt := BACnetProgramError_other;
				ELSIF stFailedFlags.bLoad THEN
					(* abort *)
					_ProgramState := BACnetProgramState_halted;
					_ReasonForHalt := BACnetProgramError_load_failed;
				ELSIF stDoneFlags.bLoad THEN
					(* DONE *)
					_bTriggerSetup := TRUE;
					_ActiveChange := BACnetProgramRequest_run;
				ELSIF (NOT _bLockedForChange) THEN
					_ReasonForHalt := BACnetProgramError_program_normal;
					CASE _ProgramChange OF
						BACnetProgramRequest_load,
						BACnetProgramRequest_run,
						BACnetProgramRequest_halt,
						BACnetProgramRequest_restart:
							(* acknowledge without execution *)
							_SetProgramReadyState	:= TRUE;
						BACnetProgramRequest_unload:
							(* execute request *)
							_ActiveChange := _ProgramChange;
					END_CASE
				END_IF

			BACnetProgramState_running:
				IF bCommonError THEN
					(* abort *)
					_ProgramState := BACnetProgramState_halted;
					_ReasonForHalt := BACnetProgramError_progerror_internal;
				ELSIF (NOT bRelease) THEN
					(* abort *)
					_ProgramState := BACnetProgramState_halted;
					_ReasonForHalt := BACnetProgramError_other;
				ELSIF bWaitForSomething THEN
					(* wait on something *)
					_ProgramState := BACnetProgramState_waiting;
				ELSIF (NOT _bLockedForChange) THEN
					_ReasonForHalt := BACnetProgramError_program_normal;
					CASE _ProgramChange OF
						BACnetProgramRequest_run:
							(* is already running *)
							_SetProgramReadyState	:= TRUE;
						BACnetProgramRequest_unload,
						BACnetProgramRequest_halt:
							(* execute request *)
							_ActiveChange := _ProgramChange;
						BACnetProgramRequest_restart,
						BACnetProgramRequest_load:
							(* retrigger setup *)
							_ActiveChange := BACnetProgramRequest_restart;
							_bTriggerSetup := TRUE;
					END_CASE
				END_IF

			BACnetProgramState_waiting:
				IF bCommonError THEN
					(* abort *)
					_ProgramState := BACnetProgramState_halted;
					_ReasonForHalt := BACnetProgramError_progerror_internal;
				ELSIF (NOT bRelease) THEN
					(* abort *)
					_ProgramState := BACnetProgramState_halted;
					_ReasonForHalt := BACnetProgramError_other;
				ELSIF (NOT bWaitForSomething) THEN
					(* got it *)
					_ProgramState := BACnetProgramState_running;
				ELSIF (NOT _bLockedForChange) THEN
					_ReasonForHalt := BACnetProgramError_program_normal;
					CASE _ProgramChange OF
						BACnetProgramRequest_run:
							(* is already running *)
							_SetProgramReadyState	:= TRUE;
						BACnetProgramRequest_unload,
						BACnetProgramRequest_halt:
							(* execute request *)
							_ActiveChange := _ProgramChange;
					END_CASE
				END_IF

			BACnetProgramState_halted:
				IF (NOT bCommonError) AND bRelease AND (NOT _bLockedForChange) THEN
					CASE _ProgramChange OF
						BACnetProgramRequest_halt:
							(* acknowledge without execution *)
							_SetProgramReadyState	:= TRUE;
						BACnetProgramRequest_unload:
							(* execute request *)
							_ActiveChange := _ProgramChange;
						BACnetProgramRequest_restart,
						BACnetProgramRequest_load:
							(* retrigger setup *)
							_ActiveChange := BACnetProgramRequest_restart;
							_bTriggerSetup := TRUE;
						BACnetProgramRequest_run:
							(* start, but don't trigger setup *)
							_ActiveChange := _ProgramChange;
							_bTriggerSetup := FALSE;
					END_CASE
				END_IF

			BACnetProgramState_unloading:
				IF bModeUnloadComplex THEN
					_ReasonForHalt := BACnetProgramError_program_normal;
					IF bCommonError THEN
						(* abort *)
						_ProgramState := BACnetProgramState_halted;
						_ActiveChange := BACnetProgramRequest_ready;
						_ReasonForHalt := BACnetProgramError_progerror_internal;
					ELSIF (NOT bRelease) THEN
						(* abort *)
						_ProgramState := BACnetProgramState_halted;
						_ActiveChange := BACnetProgramRequest_ready;
						_ReasonForHalt := BACnetProgramError_other;
					ELSIF stFailedFlags.bUnload THEN
						(* abort *)
						_ProgramState := BACnetProgramState_halted;
						_ActiveChange := BACnetProgramRequest_ready;
						_ReasonForHalt := BACnetProgramError_other;
					ELSIF stDoneFlags.bUnload THEN
						(* DONE *)
						_ActiveChange := BACnetProgramRequest_ready;
						_ProgramState := BACnetProgramState_idle;
					ELSIF (NOT _bLockedForChange) THEN
						CASE _ProgramChange OF
							BACnetProgramRequest_load,
							BACnetProgramRequest_run,
							BACnetProgramRequest_halt,
							BACnetProgramRequest_restart,
							BACnetProgramRequest_unload:
								(* acknowledge without execution *)
								_SetProgramReadyState	:= TRUE;
						END_CASE
					END_IF
				END_IF

		END_CASE
	END_IF

	(* check state of "change" request *)
	IF (_ActiveChange <> BACnetProgramRequest_ready) THEN
		(* request is active, lock execution *)
		_bLockedForChange		:= TRUE;
	ELSIF _bLockedForChange AND (NOT _SetProgramReadyState) THEN
		(* change finished, tell the stack done *)
		_SetProgramReadyState	:= TRUE;
		_bTriggerSetup			:= FALSE;
	ELSIF (_ProgramChange = BACnetProgramRequest_ready) THEN
		(* wait on new requests *)
		_SetProgramReadyState	:= FALSE;
		_bLockedForChange		:= FALSE;
		_bTriggerSetup			:= FALSE;
	ELSE
		(* new request *)
		_bTriggerSetup			:= FALSE;
	END_IF

	(* external requests *)
	stRequestFlags.bLoad			:= (_ProgramState = BACnetProgramState_loading) AND (NOT _bLockedForChange);
	stRequestFlags.bSetup			:=	(		(_ActiveChange = BACnetProgramRequest_run)
										OR	(_ActiveChange = BACnetProgramRequest_restart)
									)
								AND	_bTriggerSetup;
	stRequestFlags.bRun			:= (_ActiveChange = BACnetProgramRequest_run) AND (NOT _bTriggerSetup);
	stRequestFlags.bHalt			:= _ActiveChange = BACnetProgramRequest_halt;
	stRequestFlags.bUnload		:=	(_ActiveChange = BACnetProgramRequest_unload)
								OR	(		(_ProgramState = BACnetProgramState_unloading)
										AND	(NOT _bLockedForChange)
									);

	(* active status flags *)
	stActiveStateFlags.bIdle		:= _ProgramState = BACnetProgramState_idle;
	stActiveStateFlags.bLoading		:= _ProgramState = BACnetProgramState_loading;
	stActiveStateFlags.bRunning		:= _ProgramState = BACnetProgramState_running;
	stActiveStateFlags.bWaiting		:= _ProgramState = BACnetProgramState_waiting;
	stActiveStateFlags.bHalted		:= _ProgramState = BACnetProgramState_halted;
	stActiveStateFlags.bUnloading	:= _ProgramState = BACnetProgramState_unloading;
ELSE
	(* server device not ready, reset local ready also *)
	bReady := FALSE;
	nErrorId := BACnet_ERR_OPERATIONAL;
END_IF
(* set error flag *)
bError := (nErrorId <> BACnet_ERR_NO_ERROR);
END_FUNCTION_BLOCK

(* POU FB_BACnet_PulseConverter, ST *)
FUNCTION_BLOCK FB_BACnet_PulseConverter
VAR_IN_OUT
	Device			: FB_BACnet_Device;
END_VAR
VAR_OUTPUT
	bReady			: BOOL;
	fPresentValue	: REAL;
	nCount			: UDINT;
	bOverridden		: BOOL;
	bOutOfService	: BOOL;
	bFault			: BOOL;
	bInAlarm		: BOOL;
	bError			: BOOL;
	nErrorId		: UINT;
END_VAR
VAR
	_PresentValueIn AT%I*: REAL; 	(* ~(BACnet_PresentValue 		:		: )
								   		(BACnet_ObjectType 			: PC	: )	*)
	_Count AT%I*: UDINT;			(* ~(BACnet_Count		 		:		: ) *)
	_StatusFlags AT%I*: WORD; 		(* ~(BACnet_StatusFlags 		:		: )	*)
	_StatusFlagsBits : ST_BACnet_StatusFlags;
	_nUpdateCount : UDINT := 0;
END_VAR
(* update server device *)
IF (Device._nUpdateCount = _nUpdateCount) THEN
	Device();
END_IF
(* remind current number of update counter *)
_nUpdateCount := Device._nUpdateCount;

IF Device.bFirstCycle THEN
	(* first call of the server device since reboot/reset *)
	bReady := FALSE;

ELSIF (_StatusFlags < 4) THEN
	(* wrong mapping *)
	nErrorId := BACnet_ERR_WRONG_MAPPING;
	bReady := FALSE;

ELSIF Device.bOperational THEN
	(* ready state *)
	bReady := TRUE;
	nErrorId := BACnet_ERR_NO_ERROR;

	(* present value *)
	fPresentValue := _PresentValueIn;

	(* build bit states *)
	_StatusFlagsBits := F_BACnet_StatusFlags(_StatusFlags);

	(* copy states to output *)
	bOverridden		:= _StatusFlagsBits.overridden;
	bOutOfService	:= _StatusFlagsBits.out_of_service;
	bFault			:= _StatusFlagsBits.fault;
	bInAlarm		:= _StatusFlagsBits.in_alarm;

	(* additional information *)
	nCount			:= _Count;

ELSE
	(* server device not ready, reset local ready flag *)
	bReady := FALSE;
	nErrorId := BACnet_ERR_OPERATIONAL;
END_IF
(* set error flag *)
bError := (nErrorId <> BACnet_ERR_NO_ERROR);
END_FUNCTION_BLOCK

(* POU FB_BACnet_PulseConverter_EX, ST *)
FUNCTION_BLOCK FB_BACnet_PulseConverter_EX
VAR_IN_OUT
	Device				: FB_BACnet_Device;
END_VAR
VAR_OUTPUT
	bReady				: BOOL;
	fPresentValue		: REAL;
	bHighLimitEn		: BOOL;
	fHighLimit			: REAL;
	bLowLimitEn			: BOOL;
	fLowLimit			: REAL;
	fAdjustValue		: REAL;
	nCount				: UDINT;
	nCountBeforeChg		: UDINT;
	bOverridden			: BOOL;
	bOutOfService		: BOOL;
	bFault				: BOOL;
	bInAlarm			: BOOL;
	bOverRange			: BOOL;
	bUnderRange			: BOOL;
	bNoSensor			: BOOL;
	bOpenLoop			: BOOL;
	bShortedLoop		: BOOL;
	bCommFailure		: BOOL;
	bConfigError		: BOOL;
	bOtherFault			: BOOL;
	eEventState			: E_BACNETEVENTSTATE;
	bAckedTrans_ToOffNormal : BOOL;
	bAckedTrans_ToFault		: BOOL;
	bAckedTrans_ToNormal	: BOOL;
	tObjectID			: T_BACnet_ObjectIdentifier := 16#FFFFFFFF;
	bError				: BOOL;
	nErrorId			: UINT;
END_VAR
VAR
	_PresentValueIn AT%I*: REAL; 	(* ~(BACnet_PresentValue 		:		: )
								   		(BACnet_ObjectType 			: PC	: )	*)
	_HighLimit AT%I*: REAL;			(* ~(BACnet_HighLimit			:		: )	*)
	_LowLimit AT%I*: REAL;			(* ~(BACnet_LowLimit			:		: )	*)
	_AdjustValue AT%I*: REAL;		(* ~(BACnet_AdjustValue 		:		: ) *)
	_Count AT%I*: UDINT;			(* ~(BACnet_Count		 		:		: ) *)
	_CountBeforeChange AT%I*: UDINT;(* ~(BACnet_CountBeforeChange	:		: ) *)
	_ObjectId AT%I* : DWORD;		(* ~(BACnet_ObjectIdentifier	:		: LINK) *)
	_StatusFlags AT%I*: WORD; 		(* ~(BACnet_StatusFlags 		:		: )	*)
	_AckedTransitions AT%I*:WORD;	(* ~(BACnet_AckedTransitions	:		: ) *)
	_EventState AT%I*: WORD; 		(* ~(BACnet_EventState			:		: )	*)
	_LimitEnable AT%I*: WORD;		(* ~(BACnet_LimitEnable			:		: )	*)
	_Reliability AT%I*: WORD;		(* ~(BACnet_Reliability 		:		: )	*)
	_AckedTransBits : ST_BACnet_EventTransitionBits;
	_StatusFlagsBits : ST_BACnet_StatusFlags;
	_LimitEnableBits : ST_BACnet_LimitEnable;
	_nUpdateCount : UDINT := 0;
END_VAR
(* update server device *)
IF (Device._nUpdateCount = _nUpdateCount) THEN
	Device();
END_IF
(* remind current number of update counter *)
_nUpdateCount := Device._nUpdateCount;

IF Device.bFirstCycle THEN
	(* first call of the server device since reboot/reset *)
	bReady := FALSE;

ELSIF (F_BACnet_GetObjType(_ObjectId) <> BACnetObjectType_PulseConverter) THEN
	(* wrong mapping / invalid object ID *)
	IF _ObjectId = 0 THEN
		nErrorId := BACnet_ERR_WRONG_MAPPING;
	ELSE
		nErrorId := BACnet_ERR_INVALID_OBJECTID;
	END_IF
	bReady := FALSE;
	tObjectID := 16#FFFFFFFF;

ELSIF (_StatusFlags < 4) OR _AckedTransitions < 5 THEN
	(* wrong mapping *)
	nErrorId := BACnet_ERR_WRONG_MAPPING;
	bReady := FALSE;

ELSIF Device.bOperational THEN
	(* ready state *)
	bReady := TRUE;
	nErrorId := BACnet_ERR_NO_ERROR;

	(* present value *)
	fPresentValue := _PresentValueIn;

	(* build bit states *)
	_StatusFlagsBits := F_BACnet_StatusFlags(_StatusFlags);
	_AckedTransBits := F_BACnet_EventTransitionFlags(_AckedTransitions);
	_LimitEnableBits :=	F_BACnet_LimitEnableFlags(_LimitEnable);

	(* copy states to output *)
	bHighLimitEn:= _LimitEnableBits.highLimitEnable;
	bLowLimitEn	:= _LimitEnableBits.lowLimitEnable;
	bOverridden	:= _StatusFlagsBits.overridden;
	bOutOfService:= _StatusFlagsBits.out_of_service;
	bFault		:= _StatusFlagsBits.fault;
	bInAlarm	:= _StatusFlagsBits.in_alarm;
	bOverRange	:= (_Reliability = BACnetReliability_over_range);
	bUnderRange	:= (_Reliability = BACnetReliability_under_range);
	bNoSensor	:= (_Reliability = BACnetReliability_no_sensor);
	bOpenLoop	:= (_Reliability = BACnetReliability_open_loop);
	bShortedLoop:= (_Reliability = BACnetReliability_shorted_loop);
	bCommFailure := (_Reliability = BACnetReliability_communication_failure);
	bConfigError:= (_Reliability = BACnetReliability_configuration_error);
	bOtherFault	:= (_Reliability = BACnetReliability_unreliable_other);
	bAckedTrans_ToOffNormal := _AckedTransBits.to_offnormal;
	bAckedTrans_ToFault := _AckedTransBits.to_fault;
	bAckedTrans_ToNormal := _AckedTransBits.to_normal;

	(* convert enumeration *)
	eEventState := _EventState;

	(* additional information *)
	fHighLimit			:= _HighLimit;
	fLowLimit			:= _LowLimit;
	fAdjustValue		:= _AdjustValue;
	nCount				:= _Count;
	nCountBeforeChg		:= _CountBeforeChange;
	tObjectID		:= F_BACnet_GetObjInstance(_ObjectId);

